(* Schneider Machine Expert - Basic project ProjectX, file version 2.7.0.0 *)
(* ProjectInformations: Name=New project *)

HARDWARE
  Cpu 0: TM221CE24U
  EthernetConfiguration: NetworkName=M221, IpAllocationMode=FixedAddress, IpAddress=0.0.0.0, SubnetMask=0.0.0.0
  SerialLineConfiguration: Baud=Baud19200, Parity=ParityEven, DataBits=DataBits8, StopBits=StopBits1, PhysicalMedium=PhysicalMediumRs485, TransmissionMode=TransmissionModeModbusRtu, SlaveId=1, Addressing=SlaveAddressing
  MastTask: UsePeriodScanMode=false, PeriodScan=100
  FastTask: Period=255
  CpuBehavior: StartingMode=StartAsPreviousState, AutoSaveRamOnEeprom=true, WatchdogPeriod=250

SYMBOLS  (address, symbol, comment, settings)
  %M240     GUI_SAFE_GUARD
  %M241     GUI_START
  %M242     GUI_ACTIVE_RESET
  %M243     GUI_SET_VALUE
  %M301     SAFE_GUARD
  %M401     INIT
  %M402     BLUE_PASS
  %M403     GREEN_PASS
  %M404     SAFETY
  %M405     INPUT
  %M406     BLUE_TANK
  %M407     EXTRA_TIME_BLUE_TANK
  %M408     GREEN_TANK
  %M409     EXTRA_TIME_GREEN_TANK
  %M410     METAL_TANK
  %M411     EXTRA_TIME_METAL_TANK
  %M412     Q_FACTOR_METAL
  %M413     Q_FACTOR_METAL_I9
  %M414     Q_FACTOR_METAL_I5
  %M415     Q_FACTOR_BLUE_I9
  %M416     Q_FACTOR_BLUE_I5
  %M417     Q_FACTOR_GREEN_I9
  %M418     Q_FACTOR_GREEN_I5
  %M421     SUS
  %M422     SUSS
  %M423     SUSSS
  %M424     SUSSSS
  %M425     SUSSSSS
  %M451     START_SYS
  %M452     STOP_SYS
  %M453     STOP_SYS_HANDLE
  %M454     STOP_SYS_HANDLE2
  %M455     CLEAR_SYS_HANDLE
  %M456     STOP_HANDLE_3
  %M457     END_SYS
  %M458     STOP_HANDLE_RESET
  %M459     HANDLE_RESET_ALL
  %M460     OVER_CONDITION
  %M461     HANDLE_CHANGE_BLUE
  %M462     HANDLE_CHANGE_BLUE2
  %M463     HANDLE_CHANGE_GREEN
  %M464     HANDLE_CHANGE_GREEN2
  %M465     HANDLE_CHANGE_METAL
  %M466     HANDLE_CHANGE_METAL2
  %M501     METAL_PART
  %M502     BLUE_LINK
  %M503     GREEN_LINK
  %M504     METAL_LINK
  %M505     SET_VALUE_LINK
  %M506     TURN_OFF_SYS
  %M507     CLEAR_SYS
  %M508     TRIGGER_TURN_OFF_SYS
  %TM0        [Preset=5, Base=OneHundredMilliSeconds]
  %TM1        [Preset=15, Base=OneHundredMilliSeconds]
  %TM2        [Preset=0, Base=OneSecond]
  %TM3        [Preset=1, Base=OneSecond]
  %TM4        [Preset=0, Base=OneSecond]
  %TM5        [Preset=1, Base=OneSecond]
  %TM6        [Preset=0, Base=OneSecond]
  %TM7        [Preset=1, Base=OneSecond]
  %TM8        [Preset=2, Base=OneSecond]
  %TM9        [Preset=2, Base=OneSecond]
  %TM10       [Preset=2, Base=OneSecond]
  %TM11       [Preset=2, Base=OneSecond]
  %TM12       [Preset=2, Base=OneSecond]
  %TM13       [Preset=2, Base=OneSecond]
  %TM14       [Preset=15, Base=OneSecond]
  %TM15       [Preset=1, Base=OneSecond]
  %TM16       [Preset=40, Base=OneSecond]
  %TM17       [Preset=3, Base=OneSecond]
  %TM18       [Preset=3, Base=OneSecond]
  %TM19       [Preset=3, Base=OneSecond]
  %TM20       [Preset=3, Base=OneSecond]
  %TM21       [Preset=3, Base=OneSecond]
  %TM22       [Preset=3, Base=OneSecond]
  %C0         "Counting"
  %C1         "Dielectric"
  %C2         "Metal"
  %C3         "Blue dielec"
  %C4         "Green dielec"
  %C5         "Blue dielec (I5)"
  %C6         "Blue dielec (I9)"
  %C7         "Green dielec (I5)"
  %C8         "Green dielec (I9)"
  %C9         "Metal (I5)"
  %C10        "Metal (I9)"
  %C11        "All time count"
  %DR0        [Bits(BitForDrum(Outputs=%M301)), StepsNumber=2]

POU New POU
  (* SectionNumber=1 *)

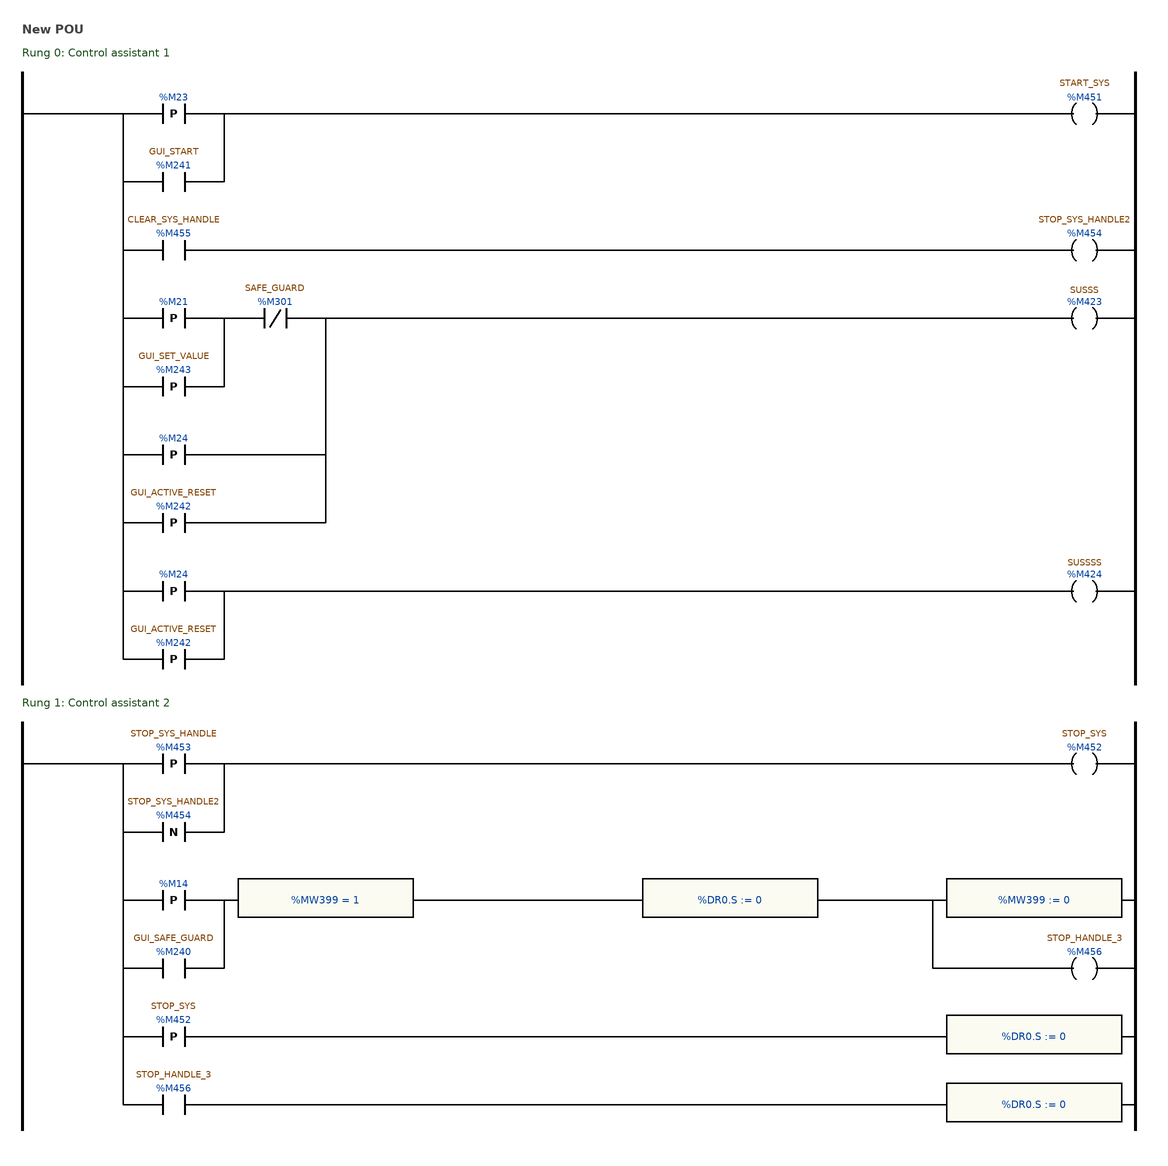

// Rung 0: Control assistant 1
  LD 1
  MPS
  AND(R %M23
  OR %M241                (* GUI_START *)
  )
  ST %M451                (* START_SYS *)
  MRD
  AND %M455               (* CLEAR_SYS_HANDLE *)
  ST %M454                (* STOP_SYS_HANDLE2 *)
  MRD
  AND(R %M21
  ORR %M243               (* GUI_SET_VALUE *)
  ANDN %M301              (* SAFE_GUARD *)
  ORR %M24
  ORR %M242               (* GUI_ACTIVE_RESET *)
  )
  ST %M423                (* SUSSS *)
  MPP
  AND(R %M24
  ORR %M242               (* GUI_ACTIVE_RESET *)
  )
  ST %M424                (* SUSSSS *)
  // as ST:
  //   START_SYS := RISING(%M23) OR GUI_START;
  //   STOP_SYS_HANDLE2 := CLEAR_SYS_HANDLE;
  //   SUSSS := (RISING(%M21) OR RISING(GUI_SET_VALUE)) AND NOT SAFE_GUARD OR RISING(%M24) OR RISING(GUI_ACTIVE_RESET);
  //   SUSSSS := RISING(%M24) OR RISING(GUI_ACTIVE_RESET);

// Rung 1: Control assistant 2
  LD 1
  MPS
  AND(R %M453             (* STOP_SYS_HANDLE *)
  ORF %M454               (* STOP_SYS_HANDLE2 *)
  )
  ST %M452                (* STOP_SYS *)
  MRD
  AND(R %M14
  OR %M240                (* GUI_SAFE_GUARD *)
  )
  AND [ %MW399 = 1 ]
  OPER [ %DR0.S := 0 ]
  [ %MW399 := 0 ]
  ST %M456                (* STOP_HANDLE_3 *)
  MRD
  ANDR %M452              (* STOP_SYS *)
  [ %DR0.S := 0 ]
  MPP
  AND %M456               (* STOP_HANDLE_3 *)
  [ %DR0.S := 0 ]
  // as ST:
  //   STOP_SYS := RISING(STOP_SYS_HANDLE) OR FALLING(STOP_SYS_HANDLE2);
  //   IF (RISING(%M14) OR GUI_SAFE_GUARD) AND %MW399 = 1 THEN %DR0.S := 0; END_IF;
  //   _t1 := (RISING(%M14) OR GUI_SAFE_GUARD) AND %MW399 = 1;
  //   IF _t1 THEN %MW399 := 0; END_IF;
  //   STOP_HANDLE_3 := _t1;
  //   IF RISING(STOP_SYS) THEN %DR0.S := 0; END_IF;
  //   IF STOP_HANDLE_3 THEN %DR0.S := 0; END_IF;

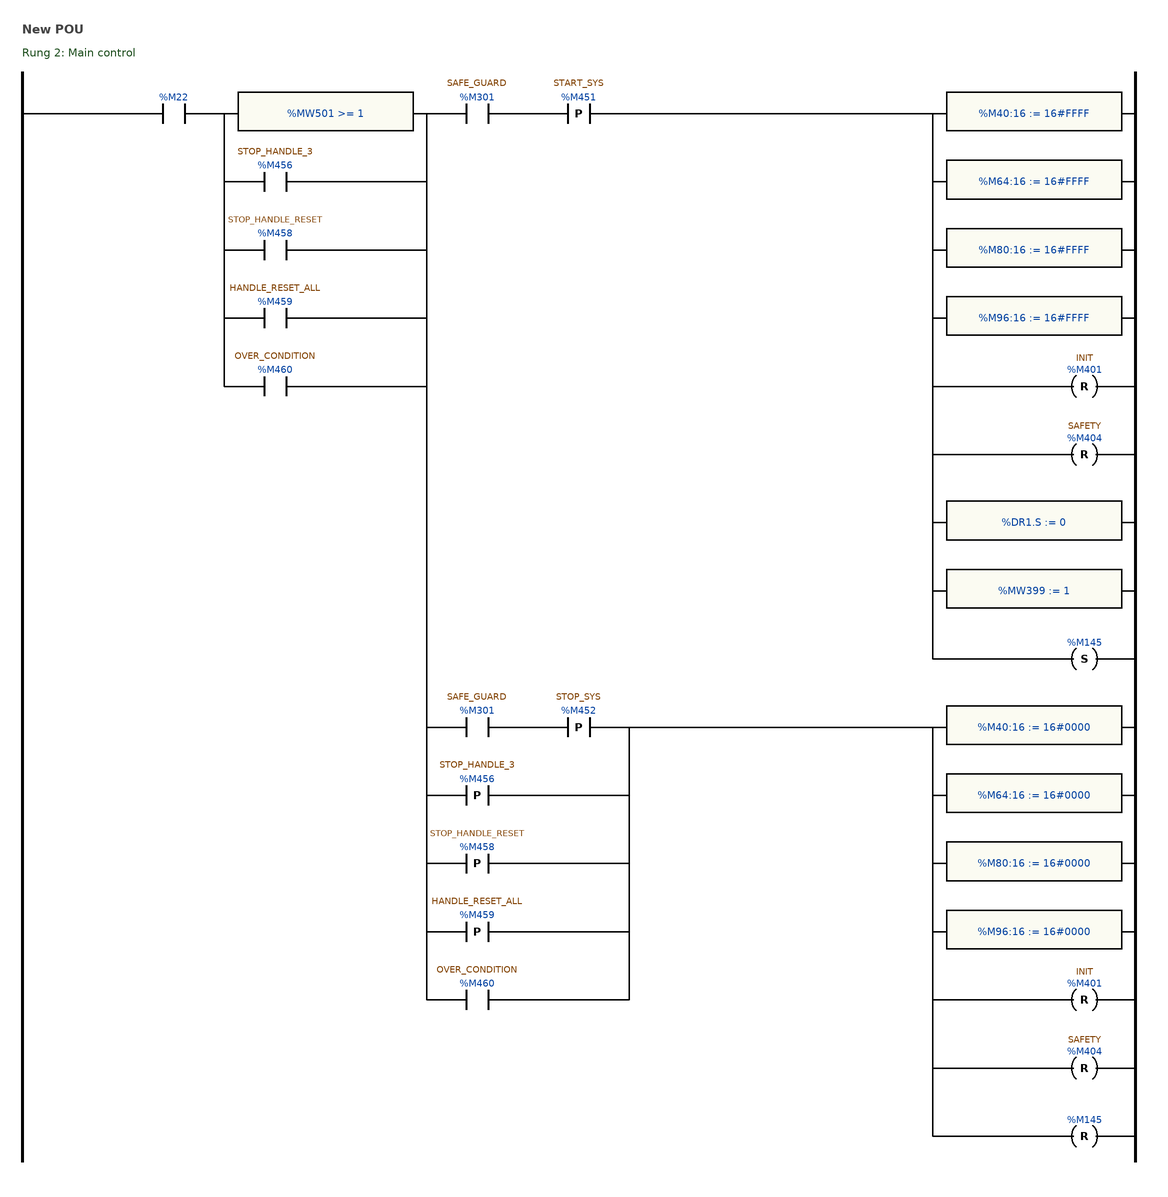

// Rung 2: Main control
  LD 1
  AND %M22
  AND( [ %MW501 >= 1 ]
  OR %M456                (* STOP_HANDLE_3 *)
  OR %M458                (* STOP_HANDLE_RESET *)
  OR %M459                (* HANDLE_RESET_ALL *)
  OR %M460                (* OVER_CONDITION *)
  )
  MPS
  AND %M301               (* SAFE_GUARD *)
  ANDR %M451              (* START_SYS *)
  [ %M40:16 := 16#FFFF ]
  [ %M64:16 := 16#FFFF ]
  [ %M80:16 := 16#FFFF ]
  [ %M96:16 := 16#FFFF ]
  R %M401                 (* INIT *)
  R %M404                 (* SAFETY *)
  [ %DR1.S := 0 ]
  [ %MW399 := 1 ]
  S %M145
  MPP
  AND( %M301              (* SAFE_GUARD *)
  ANDR %M452              (* STOP_SYS *)
  ORR %M456               (* STOP_HANDLE_3 *)
  ORR %M458               (* STOP_HANDLE_RESET *)
  ORR %M459               (* HANDLE_RESET_ALL *)
  OR %M460                (* OVER_CONDITION *)
  )
  [ %M40:16 := 16#0000 ]
  [ %M64:16 := 16#0000 ]
  [ %M80:16 := 16#0000 ]
  [ %M96:16 := 16#0000 ]
  R %M401                 (* INIT *)
  R %M404                 (* SAFETY *)
  R %M145
  // as ST:
  //   IF %M22 AND (%MW501 >= 1 OR STOP_HANDLE_3 OR STOP_HANDLE_RESET OR HANDLE_RESET_ALL OR OVER_CONDITION) AND SAFE_GUARD AND RISING(START_SYS) THEN %M40:16 := 16#FFFF; END_IF;
  //   IF %M22 AND (%MW501 >= 1 OR STOP_HANDLE_3 OR STOP_HANDLE_RESET OR HANDLE_RESET_ALL OR OVER_CONDITION) AND SAFE_GUARD AND RISING(START_SYS) THEN %M64:16 := 16#FFFF; END_IF;
  //   IF %M22 AND (%MW501 >= 1 OR STOP_HANDLE_3 OR STOP_HANDLE_RESET OR HANDLE_RESET_ALL OR OVER_CONDITION) AND SAFE_GUARD AND RISING(START_SYS) THEN %M80:16 := 16#FFFF; END_IF;
  //   IF %M22 AND (%MW501 >= 1 OR STOP_HANDLE_3 OR STOP_HANDLE_RESET OR HANDLE_RESET_ALL OR OVER_CONDITION) AND SAFE_GUARD AND RISING(START_SYS) THEN %M96:16 := 16#FFFF; END_IF;
  //   IF %M22 AND (%MW501 >= 1 OR STOP_HANDLE_3 OR STOP_HANDLE_RESET OR HANDLE_RESET_ALL OR OVER_CONDITION) AND SAFE_GUARD AND RISING(START_SYS) THEN INIT := FALSE; END_IF;
  //   IF %M22 AND (%MW501 >= 1 OR STOP_HANDLE_3 OR STOP_HANDLE_RESET OR HANDLE_RESET_ALL OR OVER_CONDITION) AND SAFE_GUARD AND RISING(START_SYS) THEN SAFETY := FALSE; END_IF;
  //   IF %M22 AND (%MW501 >= 1 OR STOP_HANDLE_3 OR STOP_HANDLE_RESET OR HANDLE_RESET_ALL OR OVER_CONDITION) AND SAFE_GUARD AND RISING(START_SYS) THEN %DR1.S := 0; END_IF;
  //   IF %M22 AND (%MW501 >= 1 OR STOP_HANDLE_3 OR STOP_HANDLE_RESET OR HANDLE_RESET_ALL OR OVER_CONDITION) AND SAFE_GUARD AND RISING(START_SYS) THEN %MW399 := 1; END_IF;
  //   IF %M22 AND (%MW501 >= 1 OR STOP_HANDLE_3 OR STOP_HANDLE_RESET OR HANDLE_RESET_ALL OR OVER_CONDITION) AND SAFE_GUARD AND RISING(START_SYS) THEN %M145 := TRUE; END_IF;
  //   IF %M22 AND (%MW501 >= 1 OR STOP_HANDLE_3 OR STOP_HANDLE_RESET OR HANDLE_RESET_ALL OR OVER_CONDITION) AND (SAFE_GUARD AND RISING(STOP_SYS) OR RISING(STOP_HANDLE_3) OR RISING(STOP_HANDLE_RESET) OR RISING(HANDLE_RESET_ALL) OR OVER_CONDITION) THEN %M40:16 := 16#0000; END_IF;
  //   IF %M22 AND (%MW501 >= 1 OR STOP_HANDLE_3 OR STOP_HANDLE_RESET OR HANDLE_RESET_ALL OR OVER_CONDITION) AND (SAFE_GUARD AND RISING(STOP_SYS) OR RISING(STOP_HANDLE_3) OR RISING(STOP_HANDLE_RESET) OR RISING(HANDLE_RESET_ALL) OR OVER_CONDITION) THEN %M64:16 := 16#0000; END_IF;
  //   IF %M22 AND (%MW501 >= 1 OR STOP_HANDLE_3 OR STOP_HANDLE_RESET OR HANDLE_RESET_ALL OR OVER_CONDITION) AND (SAFE_GUARD AND RISING(STOP_SYS) OR RISING(STOP_HANDLE_3) OR RISING(STOP_HANDLE_RESET) OR RISING(HANDLE_RESET_ALL) OR OVER_CONDITION) THEN %M80:16 := 16#0000; END_IF;
  //   IF %M22 AND (%MW501 >= 1 OR STOP_HANDLE_3 OR STOP_HANDLE_RESET OR HANDLE_RESET_ALL OR OVER_CONDITION) AND (SAFE_GUARD AND RISING(STOP_SYS) OR RISING(STOP_HANDLE_3) OR RISING(STOP_HANDLE_RESET) OR RISING(HANDLE_RESET_ALL) OR OVER_CONDITION) THEN %M96:16 := 16#0000; END_IF;
  //   IF %M22 AND (%MW501 >= 1 OR STOP_HANDLE_3 OR STOP_HANDLE_RESET OR HANDLE_RESET_ALL OR OVER_CONDITION) AND (SAFE_GUARD AND RISING(STOP_SYS) OR RISING(STOP_HANDLE_3) OR RISING(STOP_HANDLE_RESET) OR RISING(HANDLE_RESET_ALL) OR OVER_CONDITION) THEN INIT := FALSE; END_IF;
  //   IF %M22 AND (%MW501 >= 1 OR STOP_HANDLE_3 OR STOP_HANDLE_RESET OR HANDLE_RESET_ALL OR OVER_CONDITION) AND (SAFE_GUARD AND RISING(STOP_SYS) OR RISING(STOP_HANDLE_3) OR RISING(STOP_HANDLE_RESET) OR RISING(HANDLE_RESET_ALL) OR OVER_CONDITION) THEN SAFETY := FALSE; END_IF;
  //   IF %M22 AND (%MW501 >= 1 OR STOP_HANDLE_3 OR STOP_HANDLE_RESET OR HANDLE_RESET_ALL OR OVER_CONDITION) AND (SAFE_GUARD AND RISING(STOP_SYS) OR RISING(STOP_HANDLE_3) OR RISING(STOP_HANDLE_RESET) OR RISING(HANDLE_RESET_ALL) OR OVER_CONDITION) THEN %M145 := FALSE; END_IF;

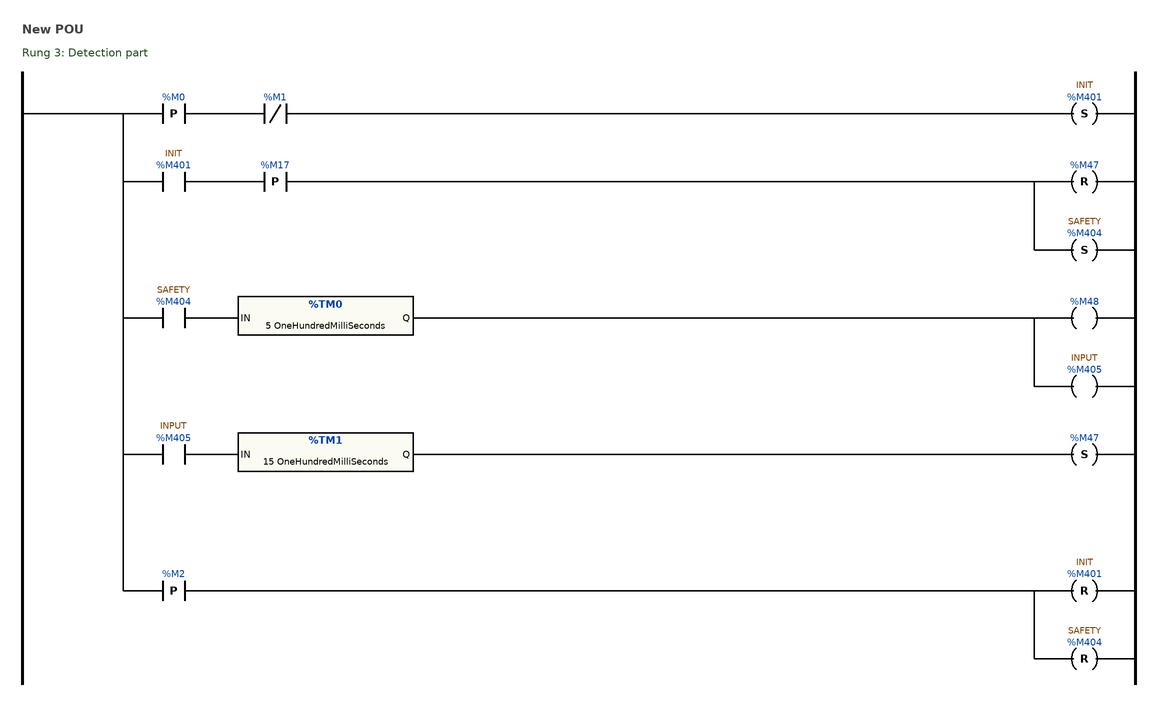

// Rung 3: Detection part
  LD 1
  MULTIFB
  LD 1
  ST %MW2009:X0
  LD %MW2009:X0
  MPS
  ANDR %M0
  ANDN %M1
  S %M401                 (* INIT *)
  MPP
  AND %M401               (* INIT *)
  ANDR %M17
  R %M47
  S %M404                 (* SAFETY *)
  BLK %TM0
  LD %MW2009:X0
  AND %M404               (* SAFETY *)
  IN
  OUT_BLK
  LD Q
  ST %M48
  ST %M405                (* INPUT *)
  END_BLK
  BLK %TM1
  LD %MW2009:X0
  AND %M405               (* INPUT *)
  IN
  OUT_BLK
  LD Q
  S %M47
  END_BLK
  LD %MW2009:X0
  ANDR %M2
  R %M401                 (* INIT *)
  R %M404                 (* SAFETY *)
  MULTIFB
  // as ST:
  //   IF RISING(%M0) AND NOT %M1 THEN INIT := TRUE; END_IF;
  //   IF INIT AND RISING(%M17) THEN %M47 := FALSE; END_IF;
  //   IF INIT AND RISING(%M17) THEN SAFETY := TRUE; END_IF;
  //   %TM0(IN := SAFETY);
  //   %M48 := %TM0.Q;
  //   INPUT := %TM0.Q;
  //   %TM1(IN := INPUT);
  //   IF %TM1.Q THEN %M47 := TRUE; END_IF;
  //   IF RISING(%M2) THEN INIT := FALSE; END_IF;
  //   IF RISING(%M2) THEN SAFETY := FALSE; END_IF;

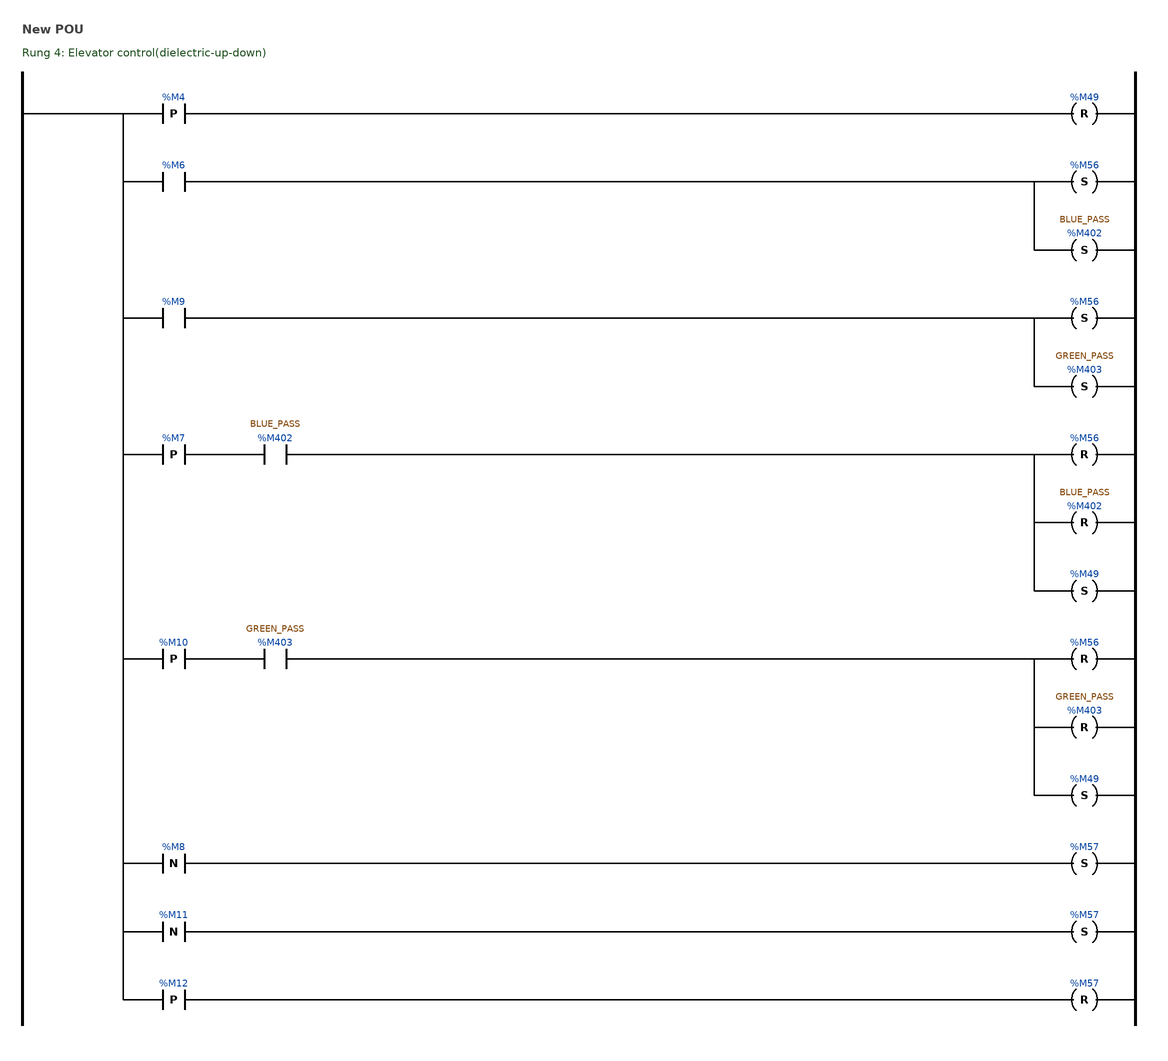

// Rung 4: Elevator control(dielectric-up-down)
  LD 1
  MPS
  ANDR %M4
  R %M49
  MRD
  AND %M6
  S %M56
  S %M402                 (* BLUE_PASS *)
  MRD
  AND %M9
  S %M56
  S %M403                 (* GREEN_PASS *)
  MRD
  ANDR %M7
  AND %M402               (* BLUE_PASS *)
  R %M56
  R %M402                 (* BLUE_PASS *)
  S %M49
  MRD
  ANDR %M10
  AND %M403               (* GREEN_PASS *)
  R %M56
  R %M403                 (* GREEN_PASS *)
  S %M49
  MRD
  ANDF %M8
  S %M57
  MRD
  ANDF %M11
  S %M57
  MPP
  ANDR %M12
  R %M57
  // as ST:
  //   IF RISING(%M4) THEN %M49 := FALSE; END_IF;
  //   IF %M6 THEN %M56 := TRUE; END_IF;
  //   IF %M6 THEN BLUE_PASS := TRUE; END_IF;
  //   IF %M9 THEN %M56 := TRUE; END_IF;
  //   IF %M9 THEN GREEN_PASS := TRUE; END_IF;
  //   IF RISING(%M7) AND BLUE_PASS THEN %M56 := FALSE; END_IF;
  //   _t1 := RISING(%M7) AND BLUE_PASS;
  //   IF _t1 THEN BLUE_PASS := FALSE; END_IF;
  //   IF _t1 THEN %M49 := TRUE; END_IF;
  //   IF RISING(%M10) AND GREEN_PASS THEN %M56 := FALSE; END_IF;
  //   _t2 := RISING(%M10) AND GREEN_PASS;
  //   IF _t2 THEN GREEN_PASS := FALSE; END_IF;
  //   IF _t2 THEN %M49 := TRUE; END_IF;
  //   IF FALLING(%M8) THEN %M57 := TRUE; END_IF;
  //   IF FALLING(%M11) THEN %M57 := TRUE; END_IF;
  //   IF RISING(%M12) THEN %M57 := FALSE; END_IF;

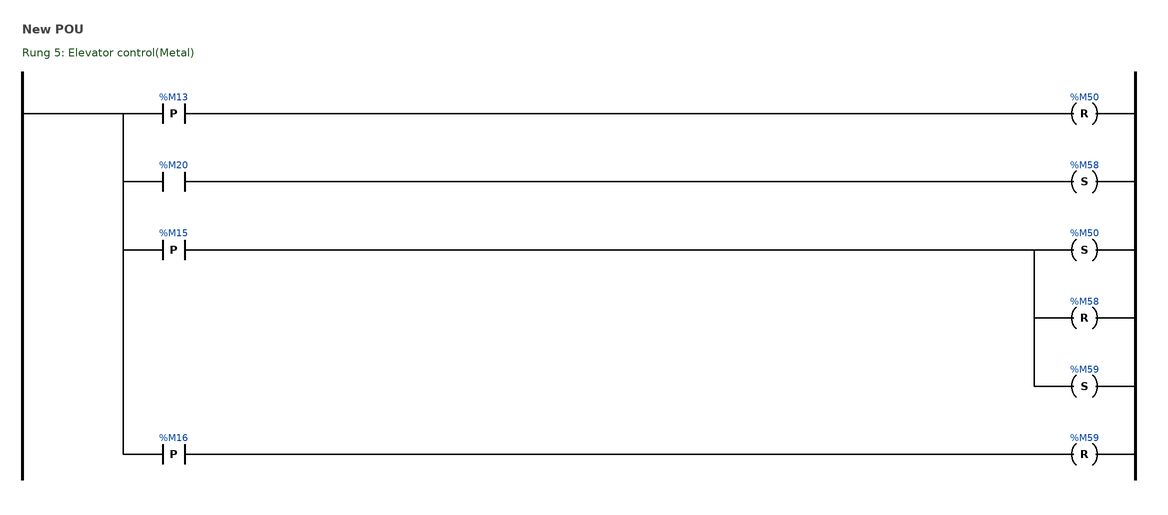

// Rung 5: Elevator control(Metal)
  LD 1
  MPS
  ANDR %M13
  R %M50
  MRD
  AND %M20
  S %M58
  MRD
  ANDR %M15
  S %M50
  R %M58
  S %M59
  MPP
  ANDR %M16
  R %M59
  // as ST:
  //   IF RISING(%M13) THEN %M50 := FALSE; END_IF;
  //   IF %M20 THEN %M58 := TRUE; END_IF;
  //   IF RISING(%M15) THEN %M50 := TRUE; END_IF;
  //   IF RISING(%M15) THEN %M58 := FALSE; END_IF;
  //   IF RISING(%M15) THEN %M59 := TRUE; END_IF;
  //   IF RISING(%M16) THEN %M59 := FALSE; END_IF;

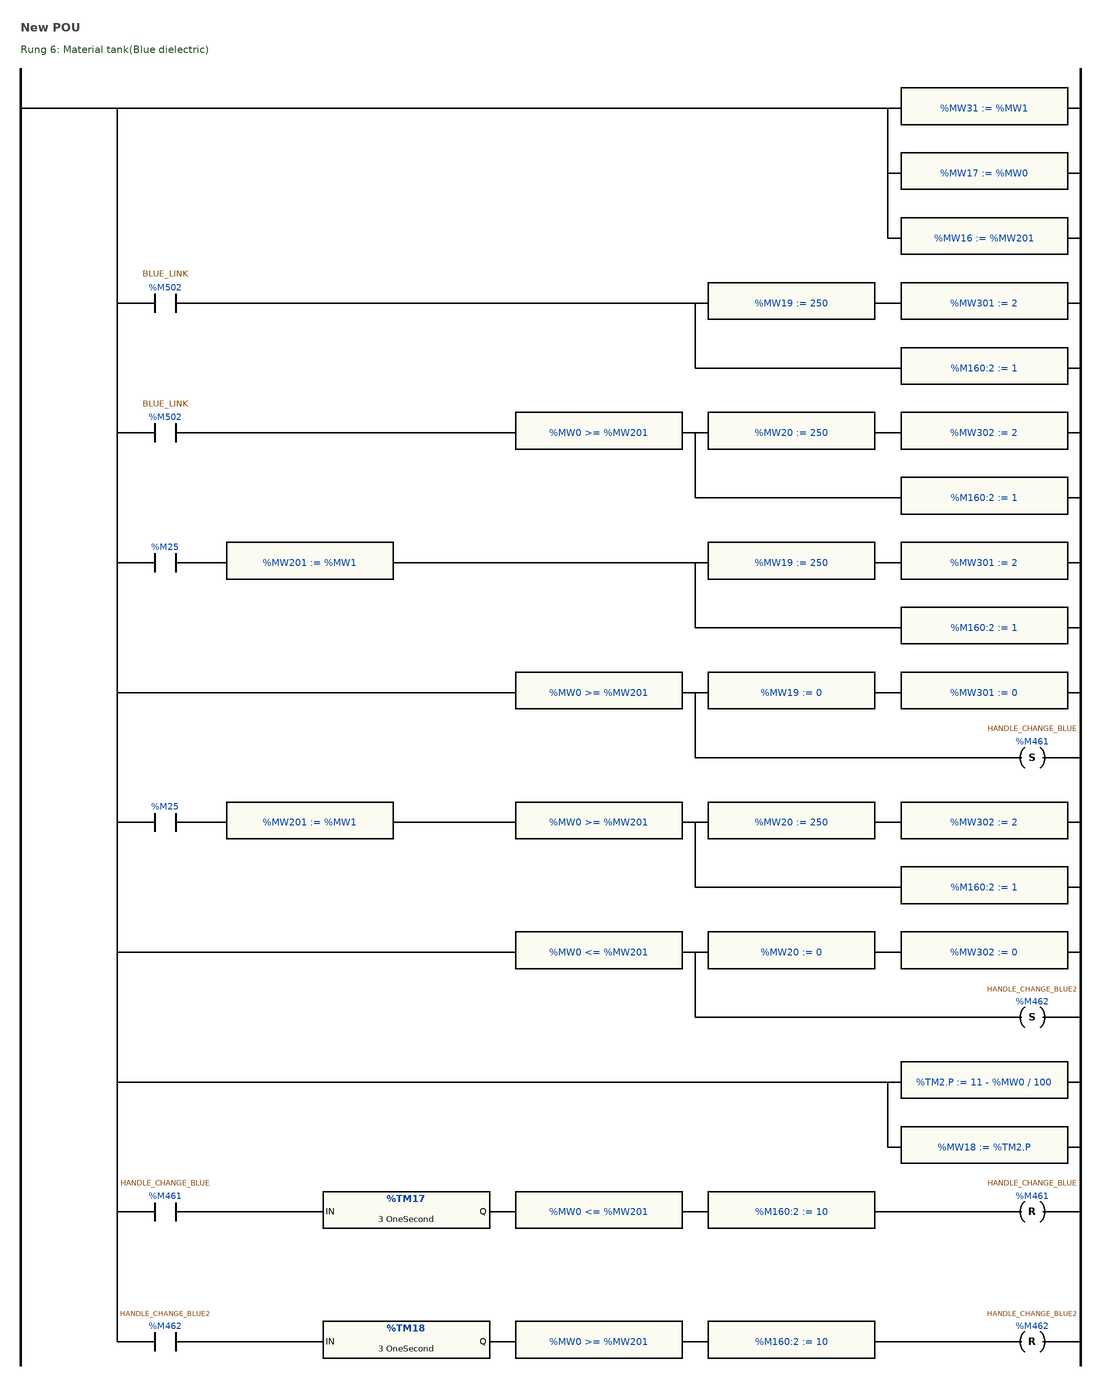

// Rung 6: Material tank(Blue dielectric)
  LD 1
  MULTIFB
  LD 1
  ST %MW2009:X0
  LD %MW2009:X0
  MPS
  [ %MW31 := %MW1 ]
  [ %MW17 := %MW0 ]
  [ %MW16 := %MW201 ]
  MRD
  AND %M502               (* BLUE_LINK *)
  MPS
  OPER [ %MW19 := 250 ]
  [ %MW301 := 2 ]
  MPP
  [ %M160:2 := 1 ]
  MRD
  AND %M502               (* BLUE_LINK *)
  AND [ %MW0 >= %MW201 ]
  MPS
  OPER [ %MW20 := 250 ]
  [ %MW302 := 2 ]
  MPP
  [ %M160:2 := 1 ]
  MRD
  AND %M25
  OPER [ %MW201 := %MW1 ]
  MPS
  OPER [ %MW19 := 250 ]
  [ %MW301 := 2 ]
  MPP
  [ %M160:2 := 1 ]
  MRD
  AND [ %MW0 >= %MW201 ]
  MPS
  OPER [ %MW19 := 0 ]
  [ %MW301 := 0 ]
  MPP
  S %M461                 (* HANDLE_CHANGE_BLUE *)
  MRD
  AND %M25
  OPER [ %MW201 := %MW1 ]
  AND [ %MW0 >= %MW201 ]
  MPS
  OPER [ %MW20 := 250 ]
  [ %MW302 := 2 ]
  MPP
  [ %M160:2 := 1 ]
  MRD
  AND [ %MW0 <= %MW201 ]
  MPS
  OPER [ %MW20 := 0 ]
  [ %MW302 := 0 ]
  MPP
  S %M462                 (* HANDLE_CHANGE_BLUE2 *)
  MPP
  [ %TM2.P := 11 - %MW0 / 100 ]
  [ %MW18 := %TM2.P ]
  BLK %TM17
  LD %MW2009:X0
  AND %M461               (* HANDLE_CHANGE_BLUE *)
  IN
  OUT_BLK
  LD Q
  AND [ %MW0 <= %MW201 ]
  OPER [ %M160:2 := 10 ]
  R %M461                 (* HANDLE_CHANGE_BLUE *)
  END_BLK
  BLK %TM18
  LD %MW2009:X0
  AND %M462               (* HANDLE_CHANGE_BLUE2 *)
  IN
  OUT_BLK
  LD Q
  AND [ %MW0 >= %MW201 ]
  OPER [ %M160:2 := 10 ]
  R %M462                 (* HANDLE_CHANGE_BLUE2 *)
  END_BLK
  MULTIFB
  // as ST:
  //   %MW31 := %MW1;
  //   %MW17 := %MW0;
  //   %MW16 := %MW201;
  //   IF BLUE_LINK THEN %MW19 := 250; END_IF;
  //   IF BLUE_LINK THEN %MW301 := 2; END_IF;
  //   IF BLUE_LINK THEN %M160:2 := 1; END_IF;
  //   IF BLUE_LINK AND %MW0 >= %MW201 THEN %MW20 := 250; END_IF;
  //   IF BLUE_LINK AND %MW0 >= %MW201 THEN %MW302 := 2; END_IF;
  //   IF BLUE_LINK AND %MW0 >= %MW201 THEN %M160:2 := 1; END_IF;
  //   IF %M25 THEN %MW201 := %MW1; END_IF;
  //   IF %M25 THEN %MW19 := 250; END_IF;
  //   IF %M25 THEN %MW301 := 2; END_IF;
  //   IF %M25 THEN %M160:2 := 1; END_IF;
  //   IF %MW0 >= %MW201 THEN %MW19 := 0; END_IF;
  //   IF %MW0 >= %MW201 THEN %MW301 := 0; END_IF;
  //   IF %MW0 >= %MW201 THEN HANDLE_CHANGE_BLUE := TRUE; END_IF;
  //   IF %M25 THEN %MW201 := %MW1; END_IF;
  //   IF %M25 AND %MW0 >= %MW201 THEN %MW20 := 250; END_IF;
  //   IF %M25 AND %MW0 >= %MW201 THEN %MW302 := 2; END_IF;
  //   IF %M25 AND %MW0 >= %MW201 THEN %M160:2 := 1; END_IF;
  //   IF %MW0 <= %MW201 THEN %MW20 := 0; END_IF;
  //   IF %MW0 <= %MW201 THEN %MW302 := 0; END_IF;
  //   IF %MW0 <= %MW201 THEN HANDLE_CHANGE_BLUE2 := TRUE; END_IF;
  //   %TM2.P := 11 - %MW0 / 100;
  //   %MW18 := %TM2.P;
  //   %TM17(IN := HANDLE_CHANGE_BLUE);
  //   IF %TM17.Q AND %MW0 <= %MW201 THEN %M160:2 := 10; END_IF;
  //   IF %TM17.Q AND %MW0 <= %MW201 THEN HANDLE_CHANGE_BLUE := FALSE; END_IF;
  //   %TM18(IN := HANDLE_CHANGE_BLUE2);
  //   IF %TM18.Q AND %MW0 >= %MW201 THEN %M160:2 := 10; END_IF;
  //   IF %TM18.Q AND %MW0 >= %MW201 THEN HANDLE_CHANGE_BLUE2 := FALSE; END_IF;

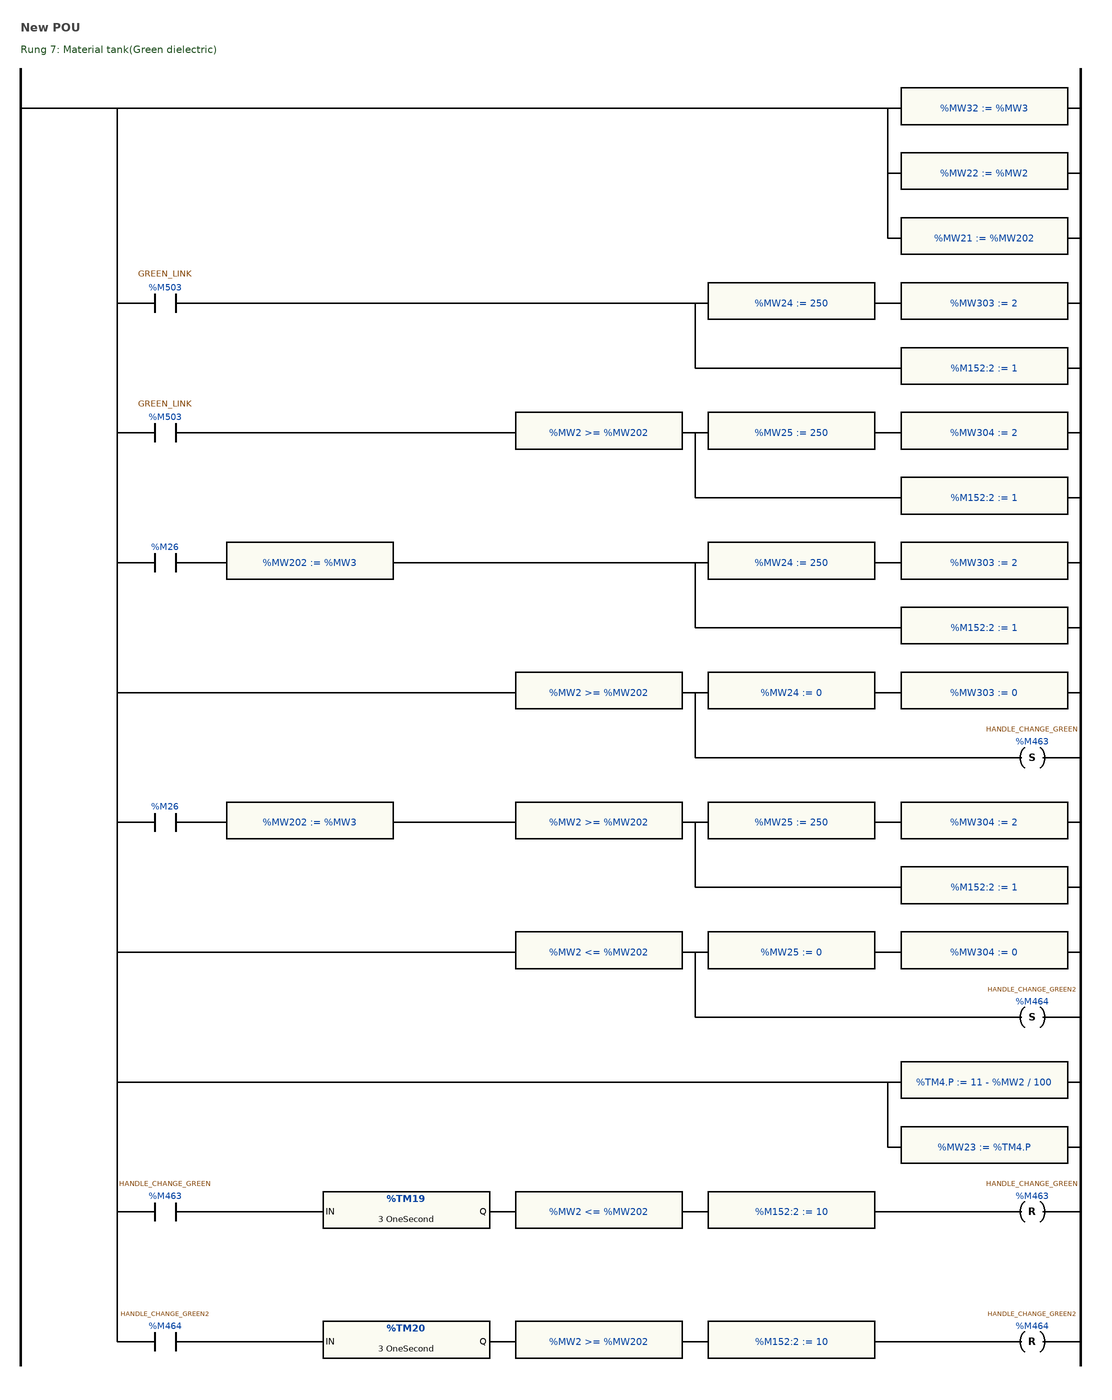

// Rung 7: Material tank(Green dielectric)
  LD 1
  MULTIFB
  LD 1
  ST %MW2009:X0
  LD %MW2009:X0
  MPS
  [ %MW32 := %MW3 ]
  [ %MW22 := %MW2 ]
  [ %MW21 := %MW202 ]
  MRD
  AND %M503               (* GREEN_LINK *)
  MPS
  OPER [ %MW24 := 250 ]
  [ %MW303 := 2 ]
  MPP
  [ %M152:2 := 1 ]
  MRD
  AND %M503               (* GREEN_LINK *)
  AND [ %MW2 >= %MW202 ]
  MPS
  OPER [ %MW25 := 250 ]
  [ %MW304 := 2 ]
  MPP
  [ %M152:2 := 1 ]
  MRD
  AND %M26
  OPER [ %MW202 := %MW3 ]
  MPS
  OPER [ %MW24 := 250 ]
  [ %MW303 := 2 ]
  MPP
  [ %M152:2 := 1 ]
  MRD
  AND [ %MW2 >= %MW202 ]
  MPS
  OPER [ %MW24 := 0 ]
  [ %MW303 := 0 ]
  MPP
  S %M463                 (* HANDLE_CHANGE_GREEN *)
  MRD
  AND %M26
  OPER [ %MW202 := %MW3 ]
  AND [ %MW2 >= %MW202 ]
  MPS
  OPER [ %MW25 := 250 ]
  [ %MW304 := 2 ]
  MPP
  [ %M152:2 := 1 ]
  MRD
  AND [ %MW2 <= %MW202 ]
  MPS
  OPER [ %MW25 := 0 ]
  [ %MW304 := 0 ]
  MPP
  S %M464                 (* HANDLE_CHANGE_GREEN2 *)
  MPP
  [ %TM4.P := 11 - %MW2 / 100 ]
  [ %MW23 := %TM4.P ]
  BLK %TM19
  LD %MW2009:X0
  AND %M463               (* HANDLE_CHANGE_GREEN *)
  IN
  OUT_BLK
  LD Q
  AND [ %MW2 <= %MW202 ]
  OPER [ %M152:2 := 10 ]
  R %M463                 (* HANDLE_CHANGE_GREEN *)
  END_BLK
  BLK %TM20
  LD %MW2009:X0
  AND %M464               (* HANDLE_CHANGE_GREEN2 *)
  IN
  OUT_BLK
  LD Q
  AND [ %MW2 >= %MW202 ]
  OPER [ %M152:2 := 10 ]
  R %M464                 (* HANDLE_CHANGE_GREEN2 *)
  END_BLK
  MULTIFB
  // as ST:
  //   %MW32 := %MW3;
  //   %MW22 := %MW2;
  //   %MW21 := %MW202;
  //   IF GREEN_LINK THEN %MW24 := 250; END_IF;
  //   IF GREEN_LINK THEN %MW303 := 2; END_IF;
  //   IF GREEN_LINK THEN %M152:2 := 1; END_IF;
  //   IF GREEN_LINK AND %MW2 >= %MW202 THEN %MW25 := 250; END_IF;
  //   IF GREEN_LINK AND %MW2 >= %MW202 THEN %MW304 := 2; END_IF;
  //   IF GREEN_LINK AND %MW2 >= %MW202 THEN %M152:2 := 1; END_IF;
  //   IF %M26 THEN %MW202 := %MW3; END_IF;
  //   IF %M26 THEN %MW24 := 250; END_IF;
  //   IF %M26 THEN %MW303 := 2; END_IF;
  //   IF %M26 THEN %M152:2 := 1; END_IF;
  //   IF %MW2 >= %MW202 THEN %MW24 := 0; END_IF;
  //   IF %MW2 >= %MW202 THEN %MW303 := 0; END_IF;
  //   IF %MW2 >= %MW202 THEN HANDLE_CHANGE_GREEN := TRUE; END_IF;
  //   IF %M26 THEN %MW202 := %MW3; END_IF;
  //   IF %M26 AND %MW2 >= %MW202 THEN %MW25 := 250; END_IF;
  //   IF %M26 AND %MW2 >= %MW202 THEN %MW304 := 2; END_IF;
  //   IF %M26 AND %MW2 >= %MW202 THEN %M152:2 := 1; END_IF;
  //   IF %MW2 <= %MW202 THEN %MW25 := 0; END_IF;
  //   IF %MW2 <= %MW202 THEN %MW304 := 0; END_IF;
  //   IF %MW2 <= %MW202 THEN HANDLE_CHANGE_GREEN2 := TRUE; END_IF;
  //   %TM4.P := 11 - %MW2 / 100;
  //   %MW23 := %TM4.P;
  //   %TM19(IN := HANDLE_CHANGE_GREEN);
  //   IF %TM19.Q AND %MW2 <= %MW202 THEN %M152:2 := 10; END_IF;
  //   IF %TM19.Q AND %MW2 <= %MW202 THEN HANDLE_CHANGE_GREEN := FALSE; END_IF;
  //   %TM20(IN := HANDLE_CHANGE_GREEN2);
  //   IF %TM20.Q AND %MW2 >= %MW202 THEN %M152:2 := 10; END_IF;
  //   IF %TM20.Q AND %MW2 >= %MW202 THEN HANDLE_CHANGE_GREEN2 := FALSE; END_IF;

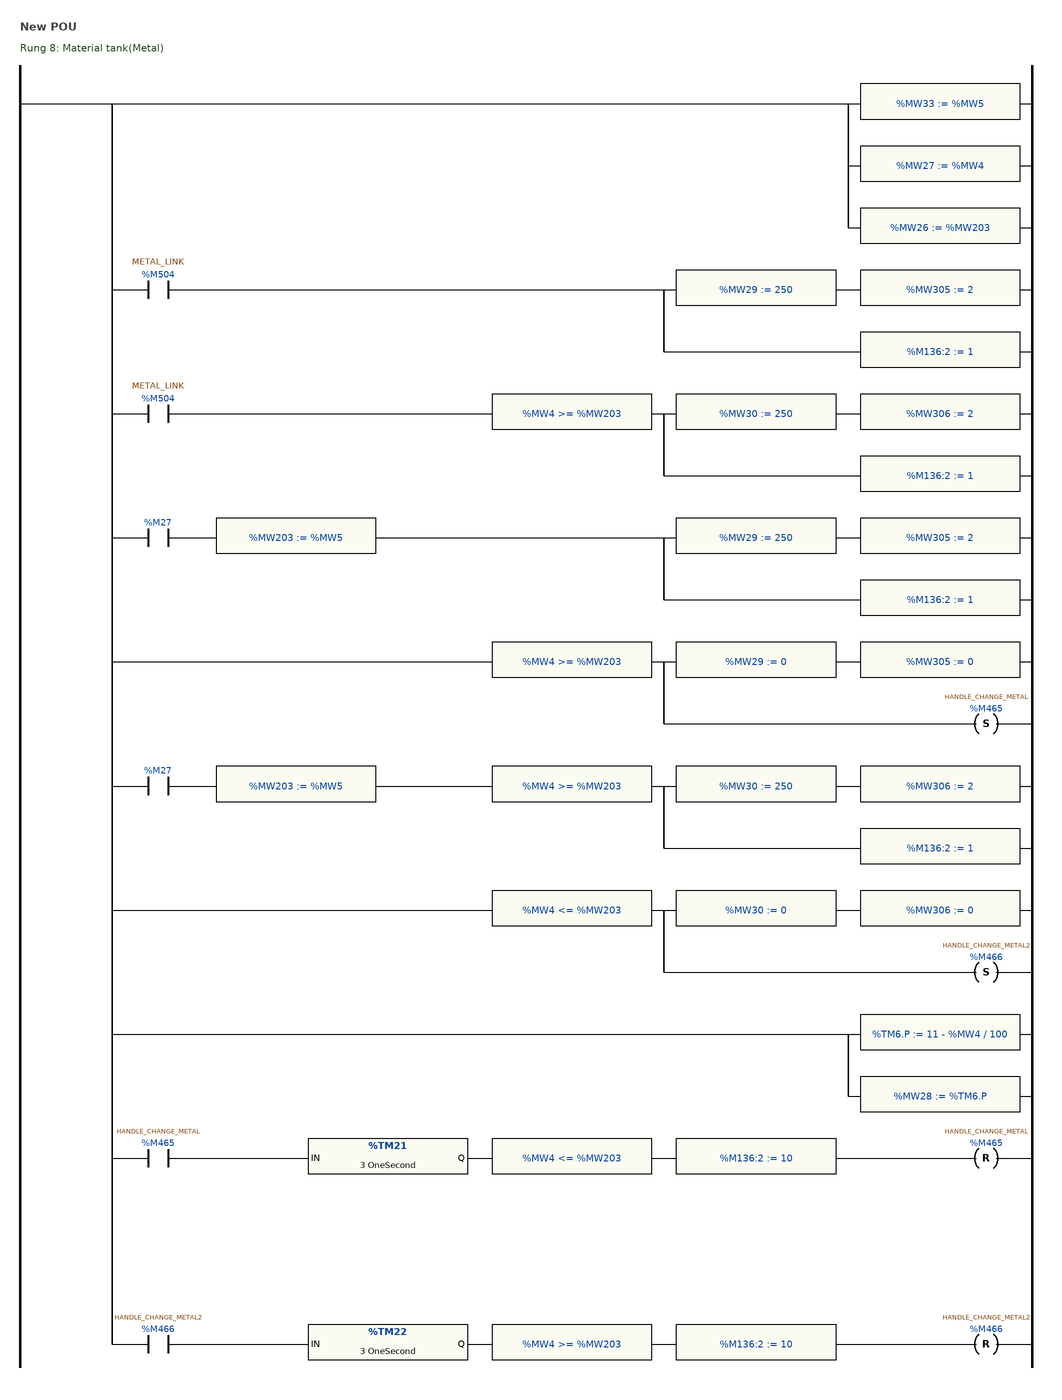

// Rung 8: Material tank(Metal)
  LD 1
  MULTIFB
  LD 1
  ST %MW2009:X0
  LD %MW2009:X0
  MPS
  [ %MW33 := %MW5 ]
  [ %MW27 := %MW4 ]
  [ %MW26 := %MW203 ]
  MRD
  AND %M504               (* METAL_LINK *)
  MPS
  OPER [ %MW29 := 250 ]
  [ %MW305 := 2 ]
  MPP
  [ %M136:2 := 1 ]
  MRD
  AND %M504               (* METAL_LINK *)
  AND [ %MW4 >= %MW203 ]
  MPS
  OPER [ %MW30 := 250 ]
  [ %MW306 := 2 ]
  MPP
  [ %M136:2 := 1 ]
  MRD
  AND %M27
  OPER [ %MW203 := %MW5 ]
  MPS
  OPER [ %MW29 := 250 ]
  [ %MW305 := 2 ]
  MPP
  [ %M136:2 := 1 ]
  MRD
  AND [ %MW4 >= %MW203 ]
  MPS
  OPER [ %MW29 := 0 ]
  [ %MW305 := 0 ]
  MPP
  S %M465                 (* HANDLE_CHANGE_METAL *)
  MRD
  AND %M27
  OPER [ %MW203 := %MW5 ]
  AND [ %MW4 >= %MW203 ]
  MPS
  OPER [ %MW30 := 250 ]
  [ %MW306 := 2 ]
  MPP
  [ %M136:2 := 1 ]
  MRD
  AND [ %MW4 <= %MW203 ]
  MPS
  OPER [ %MW30 := 0 ]
  [ %MW306 := 0 ]
  MPP
  S %M466                 (* HANDLE_CHANGE_METAL2 *)
  MPP
  [ %TM6.P := 11 - %MW4 / 100 ]
  [ %MW28 := %TM6.P ]
  BLK %TM21
  LD %MW2009:X0
  AND %M465               (* HANDLE_CHANGE_METAL *)
  IN
  OUT_BLK
  LD Q
  AND [ %MW4 <= %MW203 ]
  OPER [ %M136:2 := 10 ]
  R %M465                 (* HANDLE_CHANGE_METAL *)
  END_BLK
  BLK %TM22
  LD %MW2009:X0
  AND %M466               (* HANDLE_CHANGE_METAL2 *)
  IN
  OUT_BLK
  LD Q
  AND [ %MW4 >= %MW203 ]
  OPER [ %M136:2 := 10 ]
  R %M466                 (* HANDLE_CHANGE_METAL2 *)
  END_BLK
  MULTIFB
  // as ST:
  //   %MW33 := %MW5;
  //   %MW27 := %MW4;
  //   %MW26 := %MW203;
  //   IF METAL_LINK THEN %MW29 := 250; END_IF;
  //   IF METAL_LINK THEN %MW305 := 2; END_IF;
  //   IF METAL_LINK THEN %M136:2 := 1; END_IF;
  //   IF METAL_LINK AND %MW4 >= %MW203 THEN %MW30 := 250; END_IF;
  //   IF METAL_LINK AND %MW4 >= %MW203 THEN %MW306 := 2; END_IF;
  //   IF METAL_LINK AND %MW4 >= %MW203 THEN %M136:2 := 1; END_IF;
  //   IF %M27 THEN %MW203 := %MW5; END_IF;
  //   IF %M27 THEN %MW29 := 250; END_IF;
  //   IF %M27 THEN %MW305 := 2; END_IF;
  //   IF %M27 THEN %M136:2 := 1; END_IF;
  //   IF %MW4 >= %MW203 THEN %MW29 := 0; END_IF;
  //   IF %MW4 >= %MW203 THEN %MW305 := 0; END_IF;
  //   IF %MW4 >= %MW203 THEN HANDLE_CHANGE_METAL := TRUE; END_IF;
  //   IF %M27 THEN %MW203 := %MW5; END_IF;
  //   IF %M27 AND %MW4 >= %MW203 THEN %MW30 := 250; END_IF;
  //   IF %M27 AND %MW4 >= %MW203 THEN %MW306 := 2; END_IF;
  //   IF %M27 AND %MW4 >= %MW203 THEN %M136:2 := 1; END_IF;
  //   IF %MW4 <= %MW203 THEN %MW30 := 0; END_IF;
  //   IF %MW4 <= %MW203 THEN %MW306 := 0; END_IF;
  //   IF %MW4 <= %MW203 THEN HANDLE_CHANGE_METAL2 := TRUE; END_IF;
  //   %TM6.P := 11 - %MW4 / 100;
  //   %MW28 := %TM6.P;
  //   %TM21(IN := HANDLE_CHANGE_METAL);
  //   IF %TM21.Q AND %MW4 <= %MW203 THEN %M136:2 := 10; END_IF;
  //   IF %TM21.Q AND %MW4 <= %MW203 THEN HANDLE_CHANGE_METAL := FALSE; END_IF;
  //   %TM22(IN := HANDLE_CHANGE_METAL2);
  //   IF %TM22.Q AND %MW4 >= %MW203 THEN %M136:2 := 10; END_IF;
  //   IF %TM22.Q AND %MW4 >= %MW203 THEN HANDLE_CHANGE_METAL2 := FALSE; END_IF;

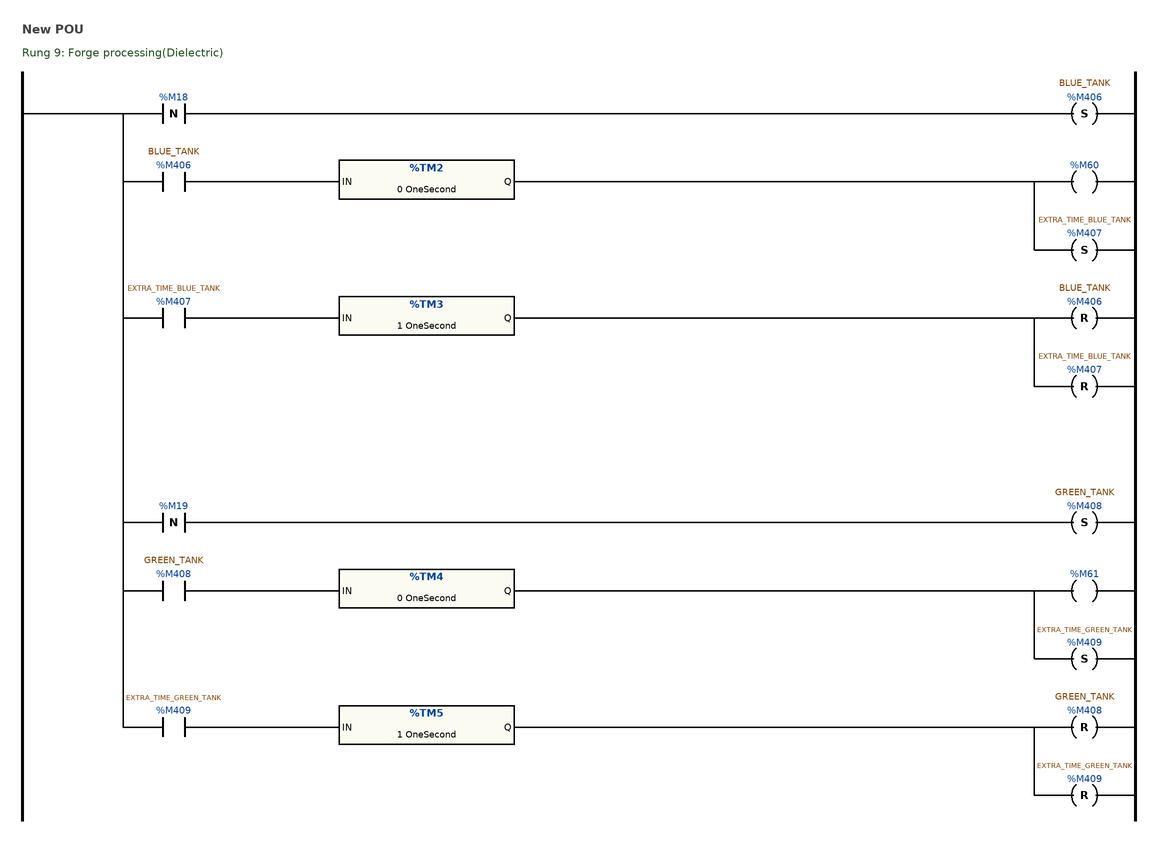

// Rung 9: Forge processing(Dielectric)
  LD 1
  MULTIFB
  LD 1
  ST %MW2009:X0
  LD %MW2009:X0
  ANDF %M18
  S %M406                 (* BLUE_TANK *)
  BLK %TM2
  LD %MW2009:X0
  AND %M406               (* BLUE_TANK *)
  IN
  OUT_BLK
  LD Q
  ST %M60
  S %M407                 (* EXTRA_TIME_BLUE_TANK *)
  END_BLK
  BLK %TM3
  LD %MW2009:X0
  AND %M407               (* EXTRA_TIME_BLUE_TANK *)
  IN
  OUT_BLK
  LD Q
  R %M406                 (* BLUE_TANK *)
  R %M407                 (* EXTRA_TIME_BLUE_TANK *)
  END_BLK
  LD %MW2009:X0
  ANDF %M19
  S %M408                 (* GREEN_TANK *)
  BLK %TM4
  LD %MW2009:X0
  AND %M408               (* GREEN_TANK *)
  IN
  OUT_BLK
  LD Q
  ST %M61
  S %M409                 (* EXTRA_TIME_GREEN_TANK *)
  END_BLK
  BLK %TM5
  LD %MW2009:X0
  AND %M409               (* EXTRA_TIME_GREEN_TANK *)
  IN
  OUT_BLK
  LD Q
  R %M408                 (* GREEN_TANK *)
  R %M409                 (* EXTRA_TIME_GREEN_TANK *)
  END_BLK
  MULTIFB
  // as ST:
  //   IF FALLING(%M18) THEN BLUE_TANK := TRUE; END_IF;
  //   %TM2(IN := BLUE_TANK);
  //   %M60 := %TM2.Q;
  //   IF %TM2.Q THEN EXTRA_TIME_BLUE_TANK := TRUE; END_IF;
  //   %TM3(IN := EXTRA_TIME_BLUE_TANK);
  //   IF %TM3.Q THEN BLUE_TANK := FALSE; END_IF;
  //   IF %TM3.Q THEN EXTRA_TIME_BLUE_TANK := FALSE; END_IF;
  //   IF FALLING(%M19) THEN GREEN_TANK := TRUE; END_IF;
  //   %TM4(IN := GREEN_TANK);
  //   %M61 := %TM4.Q;
  //   IF %TM4.Q THEN EXTRA_TIME_GREEN_TANK := TRUE; END_IF;
  //   %TM5(IN := EXTRA_TIME_GREEN_TANK);
  //   IF %TM5.Q THEN GREEN_TANK := FALSE; END_IF;
  //   IF %TM5.Q THEN EXTRA_TIME_GREEN_TANK := FALSE; END_IF;

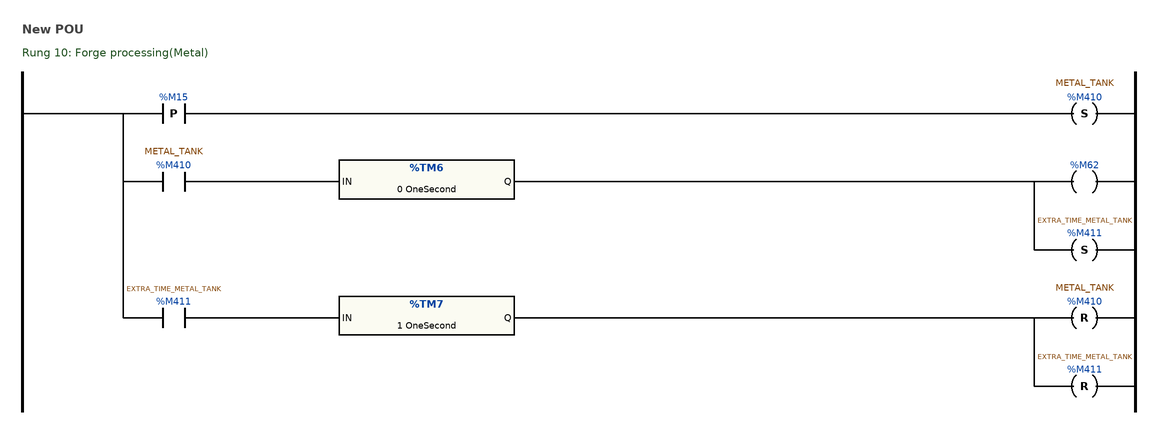

// Rung 10: Forge processing(Metal)
  LD 1
  MULTIFB
  LD 1
  ST %MW2009:X0
  LD %MW2009:X0
  ANDR %M15
  S %M410                 (* METAL_TANK *)
  BLK %TM6
  LD %MW2009:X0
  AND %M410               (* METAL_TANK *)
  IN
  OUT_BLK
  LD Q
  ST %M62
  S %M411                 (* EXTRA_TIME_METAL_TANK *)
  END_BLK
  BLK %TM7
  LD %MW2009:X0
  AND %M411               (* EXTRA_TIME_METAL_TANK *)
  IN
  OUT_BLK
  LD Q
  R %M410                 (* METAL_TANK *)
  R %M411                 (* EXTRA_TIME_METAL_TANK *)
  END_BLK
  MULTIFB
  // as ST:
  //   IF RISING(%M15) THEN METAL_TANK := TRUE; END_IF;
  //   %TM6(IN := METAL_TANK);
  //   %M62 := %TM6.Q;
  //   IF %TM6.Q THEN EXTRA_TIME_METAL_TANK := TRUE; END_IF;
  //   %TM7(IN := EXTRA_TIME_METAL_TANK);
  //   IF %TM7.Q THEN METAL_TANK := FALSE; END_IF;
  //   IF %TM7.Q THEN EXTRA_TIME_METAL_TANK := FALSE; END_IF;

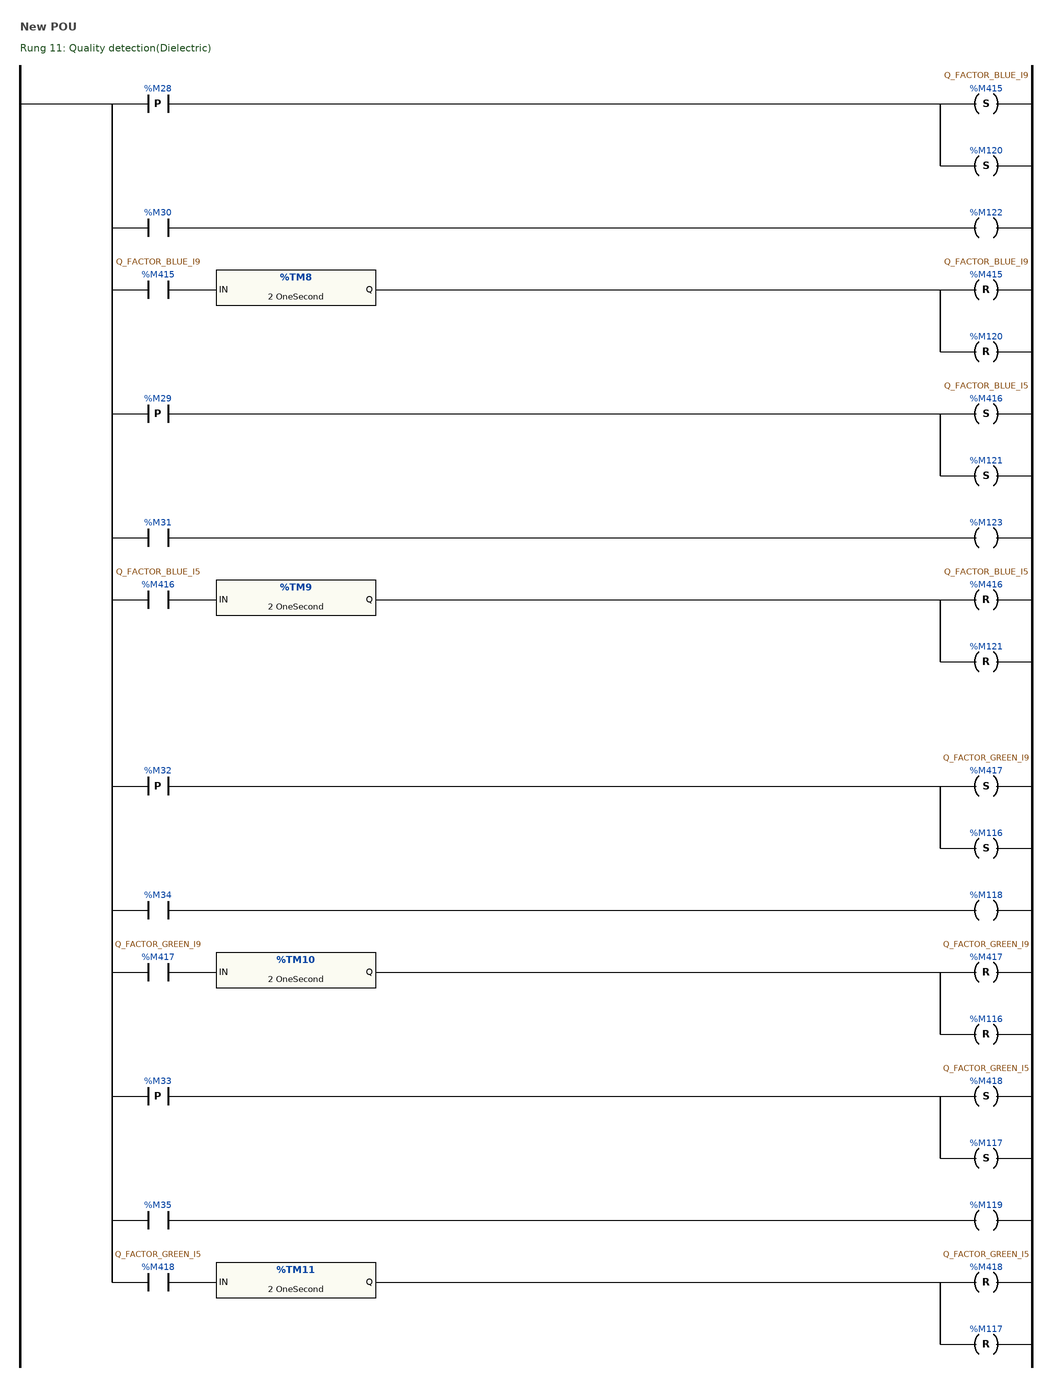

// Rung 11: Quality detection(Dielectric)
  LD 1
  MULTIFB
  LD 1
  ST %MW2009:X0
  LD %MW2009:X0
  MPS
  ANDR %M28
  S %M415                 (* Q_FACTOR_BLUE_I9 *)
  S %M120
  MPP
  AND %M30
  ST %M122
  BLK %TM8
  LD %MW2009:X0
  AND %M415               (* Q_FACTOR_BLUE_I9 *)
  IN
  OUT_BLK
  LD Q
  R %M415                 (* Q_FACTOR_BLUE_I9 *)
  R %M120
  END_BLK
  LD %MW2009:X0
  MPS
  ANDR %M29
  S %M416                 (* Q_FACTOR_BLUE_I5 *)
  S %M121
  MPP
  AND %M31
  ST %M123
  BLK %TM9
  LD %MW2009:X0
  AND %M416               (* Q_FACTOR_BLUE_I5 *)
  IN
  OUT_BLK
  LD Q
  R %M416                 (* Q_FACTOR_BLUE_I5 *)
  R %M121
  END_BLK
  LD %MW2009:X0
  MPS
  ANDR %M32
  S %M417                 (* Q_FACTOR_GREEN_I9 *)
  S %M116
  MPP
  AND %M34
  ST %M118
  BLK %TM10
  LD %MW2009:X0
  AND %M417               (* Q_FACTOR_GREEN_I9 *)
  IN
  OUT_BLK
  LD Q
  R %M417                 (* Q_FACTOR_GREEN_I9 *)
  R %M116
  END_BLK
  LD %MW2009:X0
  MPS
  ANDR %M33
  S %M418                 (* Q_FACTOR_GREEN_I5 *)
  S %M117
  MPP
  AND %M35
  ST %M119
  BLK %TM11
  LD %MW2009:X0
  AND %M418               (* Q_FACTOR_GREEN_I5 *)
  IN
  OUT_BLK
  LD Q
  R %M418                 (* Q_FACTOR_GREEN_I5 *)
  R %M117
  END_BLK
  MULTIFB
  // as ST:
  //   IF RISING(%M28) THEN Q_FACTOR_BLUE_I9 := TRUE; END_IF;
  //   IF RISING(%M28) THEN %M120 := TRUE; END_IF;
  //   %M122 := %M30;
  //   %TM8(IN := Q_FACTOR_BLUE_I9);
  //   IF %TM8.Q THEN Q_FACTOR_BLUE_I9 := FALSE; END_IF;
  //   IF %TM8.Q THEN %M120 := FALSE; END_IF;
  //   IF RISING(%M29) THEN Q_FACTOR_BLUE_I5 := TRUE; END_IF;
  //   IF RISING(%M29) THEN %M121 := TRUE; END_IF;
  //   %M123 := %M31;
  //   %TM9(IN := Q_FACTOR_BLUE_I5);
  //   IF %TM9.Q THEN Q_FACTOR_BLUE_I5 := FALSE; END_IF;
  //   IF %TM9.Q THEN %M121 := FALSE; END_IF;
  //   IF RISING(%M32) THEN Q_FACTOR_GREEN_I9 := TRUE; END_IF;
  //   IF RISING(%M32) THEN %M116 := TRUE; END_IF;
  //   %M118 := %M34;
  //   %TM10(IN := Q_FACTOR_GREEN_I9);
  //   IF %TM10.Q THEN Q_FACTOR_GREEN_I9 := FALSE; END_IF;
  //   IF %TM10.Q THEN %M116 := FALSE; END_IF;
  //   IF RISING(%M33) THEN Q_FACTOR_GREEN_I5 := TRUE; END_IF;
  //   IF RISING(%M33) THEN %M117 := TRUE; END_IF;
  //   %M119 := %M35;
  //   %TM11(IN := Q_FACTOR_GREEN_I5);
  //   IF %TM11.Q THEN Q_FACTOR_GREEN_I5 := FALSE; END_IF;
  //   IF %TM11.Q THEN %M117 := FALSE; END_IF;

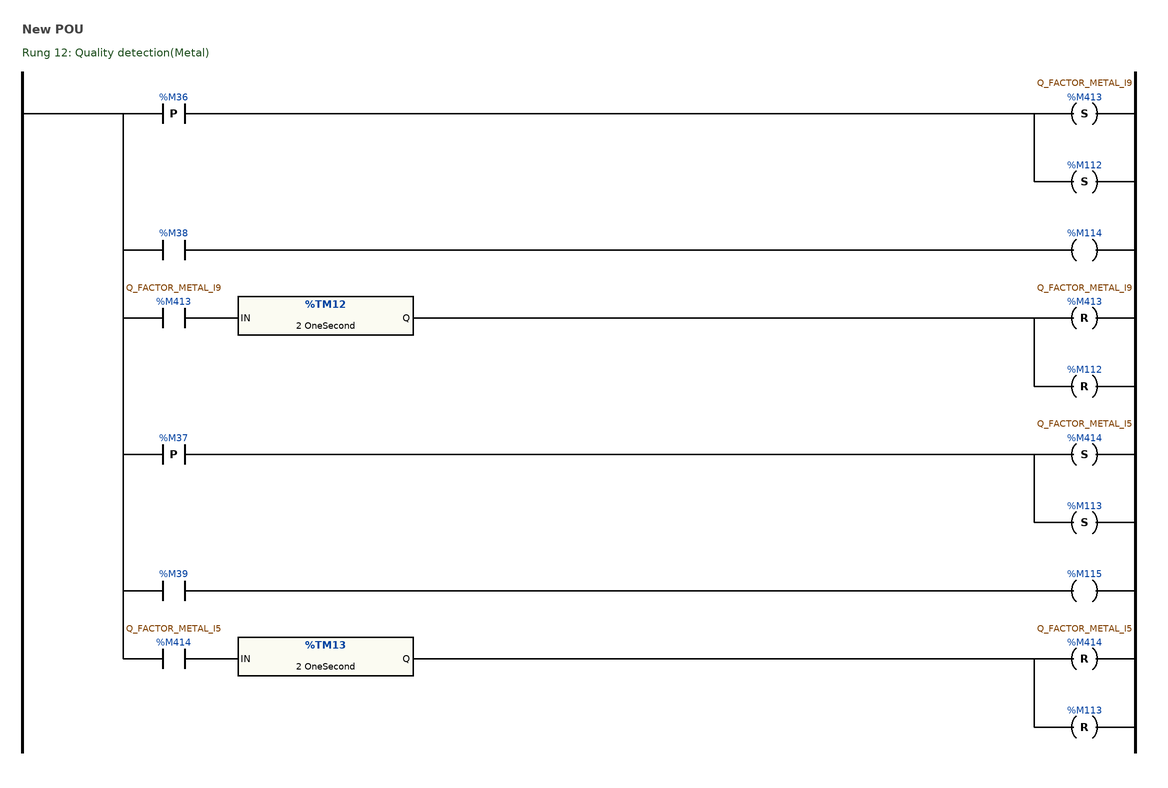

// Rung 12: Quality detection(Metal)
  LD 1
  MULTIFB
  LD 1
  ST %MW2009:X0
  LD %MW2009:X0
  MPS
  ANDR %M36
  S %M413                 (* Q_FACTOR_METAL_I9 *)
  S %M112
  MPP
  AND %M38
  ST %M114
  BLK %TM12
  LD %MW2009:X0
  AND %M413               (* Q_FACTOR_METAL_I9 *)
  IN
  OUT_BLK
  LD Q
  R %M413                 (* Q_FACTOR_METAL_I9 *)
  R %M112
  END_BLK
  LD %MW2009:X0
  MPS
  ANDR %M37
  S %M414                 (* Q_FACTOR_METAL_I5 *)
  S %M113
  MPP
  AND %M39
  ST %M115
  BLK %TM13
  LD %MW2009:X0
  AND %M414               (* Q_FACTOR_METAL_I5 *)
  IN
  OUT_BLK
  LD Q
  R %M414                 (* Q_FACTOR_METAL_I5 *)
  R %M113
  END_BLK
  MULTIFB
  // as ST:
  //   IF RISING(%M36) THEN Q_FACTOR_METAL_I9 := TRUE; END_IF;
  //   IF RISING(%M36) THEN %M112 := TRUE; END_IF;
  //   %M114 := %M38;
  //   %TM12(IN := Q_FACTOR_METAL_I9);
  //   IF %TM12.Q THEN Q_FACTOR_METAL_I9 := FALSE; END_IF;
  //   IF %TM12.Q THEN %M112 := FALSE; END_IF;
  //   IF RISING(%M37) THEN Q_FACTOR_METAL_I5 := TRUE; END_IF;
  //   IF RISING(%M37) THEN %M113 := TRUE; END_IF;
  //   %M115 := %M39;
  //   %TM13(IN := Q_FACTOR_METAL_I5);
  //   IF %TM13.Q THEN Q_FACTOR_METAL_I5 := FALSE; END_IF;
  //   IF %TM13.Q THEN %M113 := FALSE; END_IF;

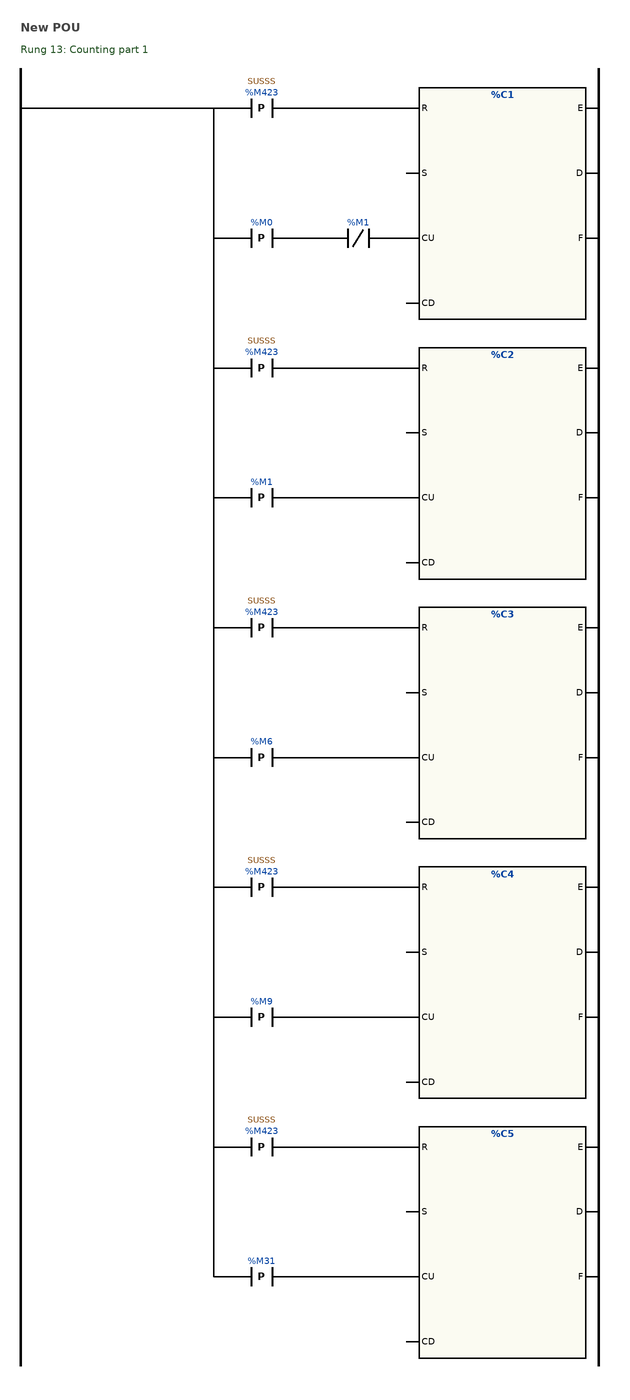

// Rung 13: Counting part 1
  LD 1
  MULTIFB
  LD 1
  ST %MW2009:X0
  BLK %C1
  LD %MW2009:X0
  MPS
  ANDR %M423              (* SUSSS *)
  R
  MPP
  ANDR %M0
  ANDN %M1
  CU
  END_BLK
  BLK %C2
  LD %MW2009:X0
  MPS
  ANDR %M423              (* SUSSS *)
  R
  MPP
  ANDR %M1
  CU
  END_BLK
  BLK %C3
  LD %MW2009:X0
  MPS
  ANDR %M423              (* SUSSS *)
  R
  MPP
  ANDR %M6
  CU
  END_BLK
  BLK %C4
  LD %MW2009:X0
  MPS
  ANDR %M423              (* SUSSS *)
  R
  MPP
  ANDR %M9
  CU
  END_BLK
  BLK %C5
  LD %MW2009:X0
  MPS
  ANDR %M423              (* SUSSS *)
  R
  MPP
  ANDR %M31
  CU
  END_BLK
  MULTIFB
  // as ST:
  //   %C1(R := RISING(SUSSS), CU := RISING(%M0) AND NOT %M1);
  //   %C2(R := RISING(SUSSS), CU := RISING(%M1));
  //   %C3(R := RISING(SUSSS), CU := RISING(%M6));
  //   %C4(R := RISING(SUSSS), CU := RISING(%M9));
  //   %C5(R := RISING(SUSSS), CU := RISING(%M31));

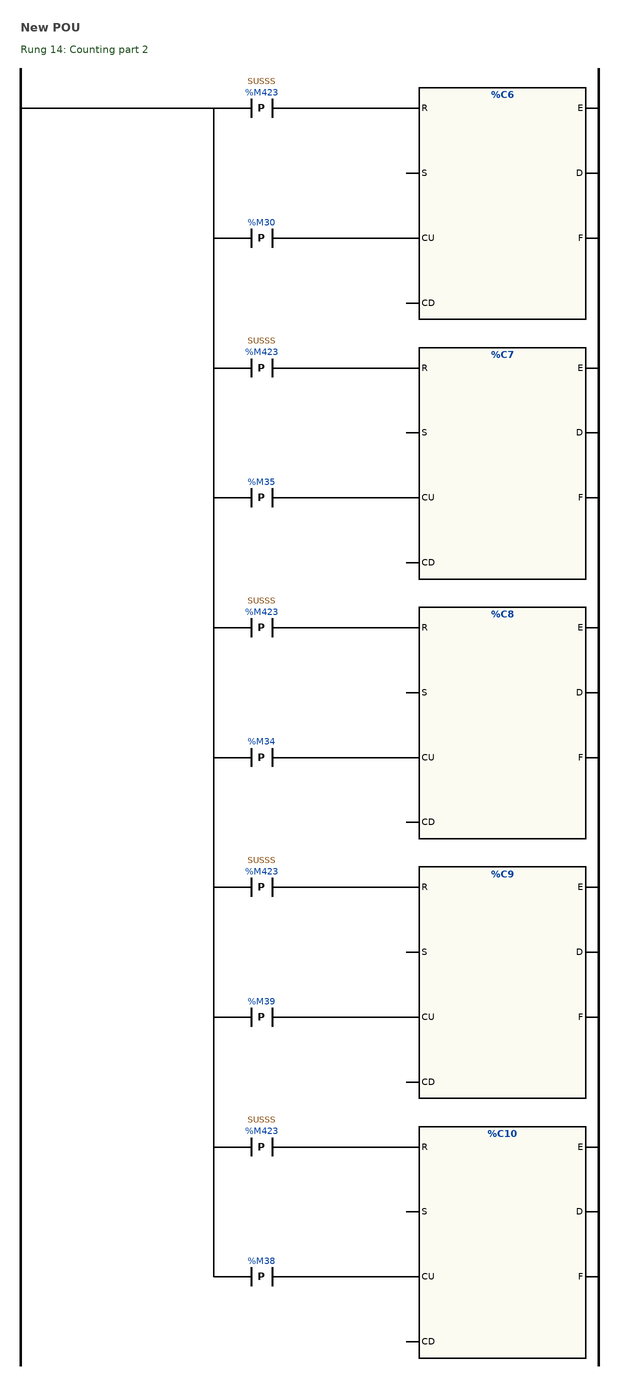

// Rung 14: Counting part 2
  LD 1
  MULTIFB
  LD 1
  ST %MW2009:X0
  BLK %C6
  LD %MW2009:X0
  MPS
  ANDR %M423              (* SUSSS *)
  R
  MPP
  ANDR %M30
  CU
  END_BLK
  BLK %C7
  LD %MW2009:X0
  MPS
  ANDR %M423              (* SUSSS *)
  R
  MPP
  ANDR %M35
  CU
  END_BLK
  BLK %C8
  LD %MW2009:X0
  MPS
  ANDR %M423              (* SUSSS *)
  R
  MPP
  ANDR %M34
  CU
  END_BLK
  BLK %C9
  LD %MW2009:X0
  MPS
  ANDR %M423              (* SUSSS *)
  R
  MPP
  ANDR %M39
  CU
  END_BLK
  BLK %C10
  LD %MW2009:X0
  MPS
  ANDR %M423              (* SUSSS *)
  R
  MPP
  ANDR %M38
  CU
  END_BLK
  MULTIFB
  // as ST:
  //   %C6(R := RISING(SUSSS), CU := RISING(%M30));
  //   %C7(R := RISING(SUSSS), CU := RISING(%M35));
  //   %C8(R := RISING(SUSSS), CU := RISING(%M34));
  //   %C9(R := RISING(SUSSS), CU := RISING(%M39));
  //   %C10(R := RISING(SUSSS), CU := RISING(%M38));

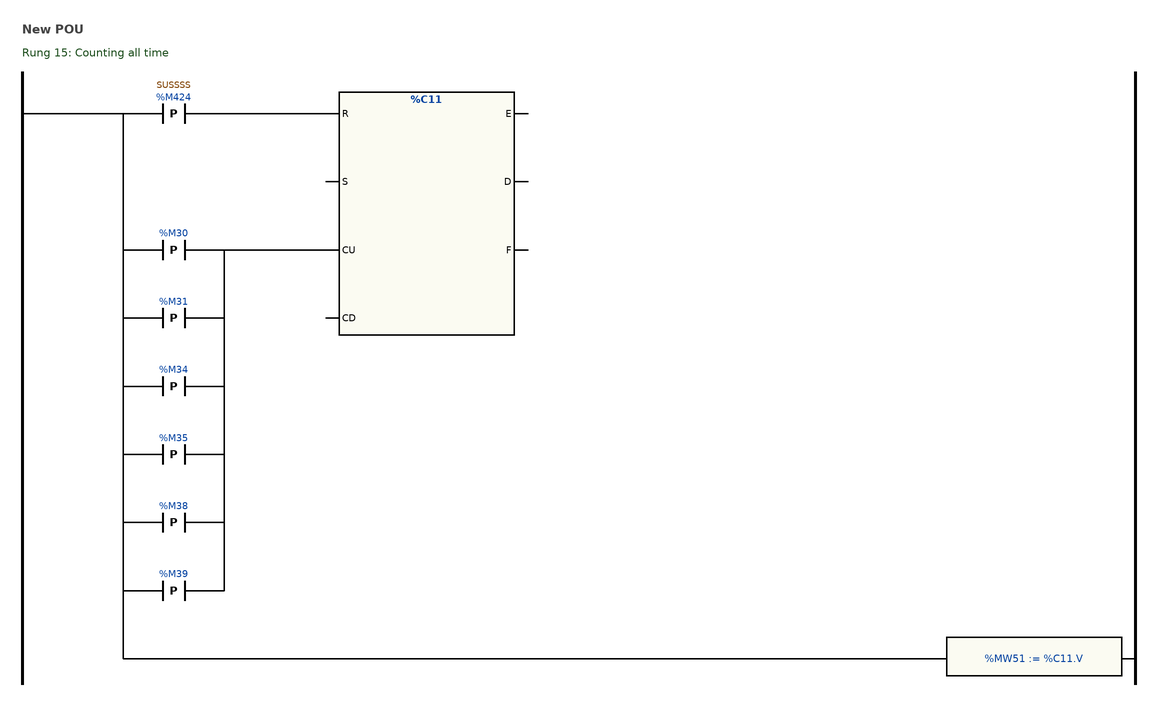

// Rung 15: Counting all time
  LD 1
  MULTIFB
  LD 1
  ST %MW2009:X0
  BLK %C11
  LD %MW2009:X0
  MPS
  ANDR %M424              (* SUSSSS *)
  R
  MPP
  AND(R %M30
  ORR %M31
  ORR %M34
  ORR %M35
  ORR %M38
  ORR %M39
  )
  CU
  END_BLK
  LD %MW2009:X0
  [ %MW51 := %C11.V ]
  MULTIFB
  // as ST:
  //   %C11(R := RISING(SUSSSS), CU := RISING(%M30) OR RISING(%M31) OR RISING(%M34) OR RISING(%M35) OR RISING(%M38) OR RISING(%M39));
  //   %MW51 := %C11.V;

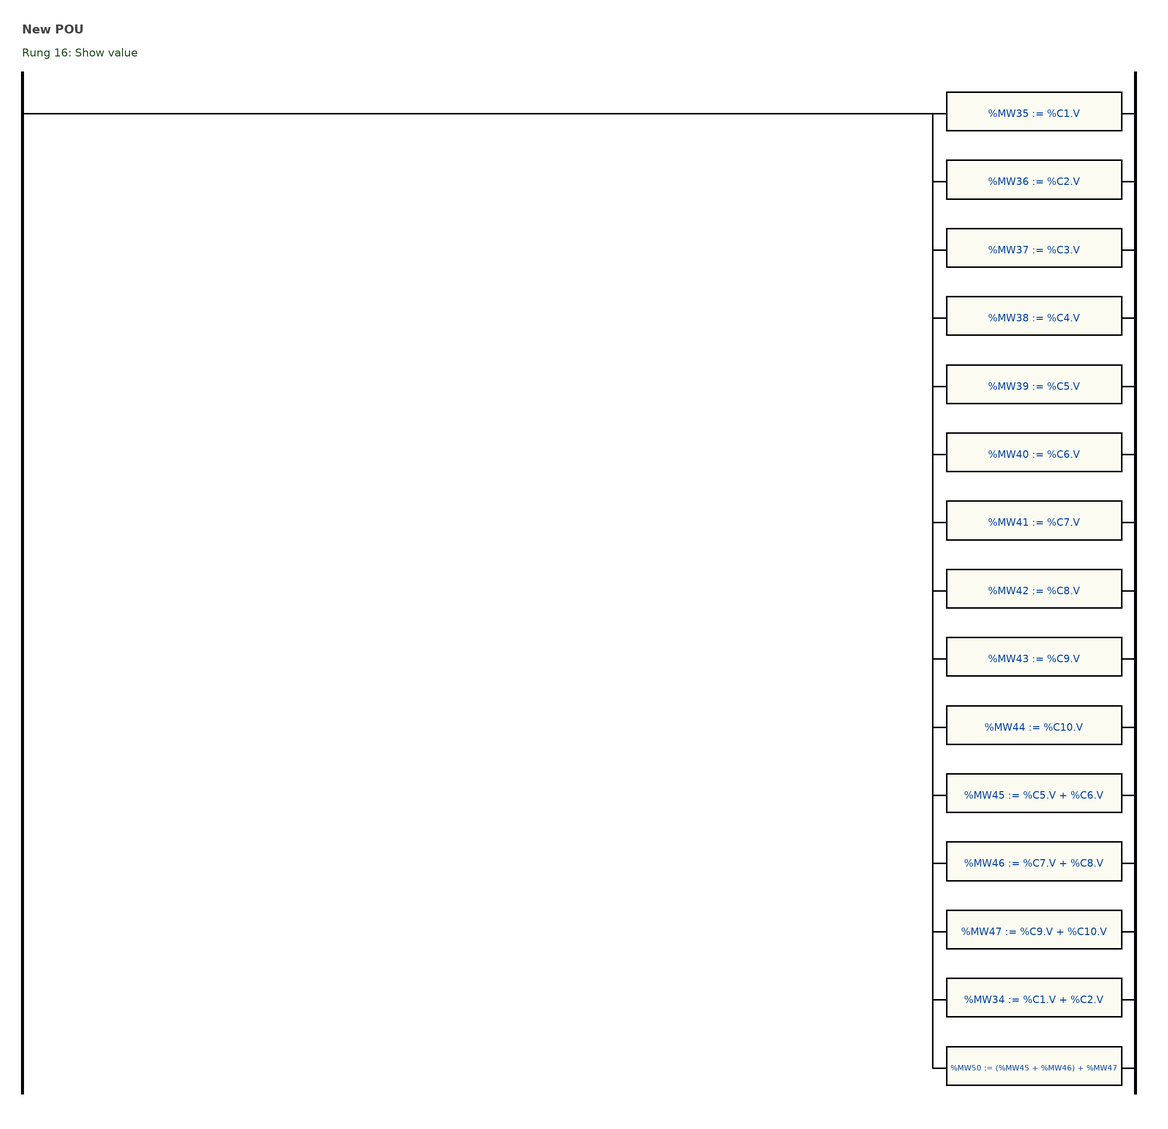

// Rung 16: Show value
  LD 1
  [ %MW35 := %C1.V ]
  [ %MW36 := %C2.V ]
  [ %MW37 := %C3.V ]
  [ %MW38 := %C4.V ]
  [ %MW39 := %C5.V ]
  [ %MW40 := %C6.V ]
  [ %MW41 := %C7.V ]
  [ %MW42 := %C8.V ]
  [ %MW43 := %C9.V ]
  [ %MW44 := %C10.V ]
  [ %MW45 := %C5.V + %C6.V ]
  [ %MW46 := %C7.V + %C8.V ]
  [ %MW47 := %C9.V + %C10.V ]
  [ %MW34 := %C1.V + %C2.V ]
  [ %MW50 := ( %MW45 + %MW46 ) + %MW47 ]
  // as ST:
  //   %MW35 := %C1.V;
  //   %MW36 := %C2.V;
  //   %MW37 := %C3.V;
  //   %MW38 := %C4.V;
  //   %MW39 := %C5.V;
  //   %MW40 := %C6.V;
  //   %MW41 := %C7.V;
  //   %MW42 := %C8.V;
  //   %MW43 := %C9.V;
  //   %MW44 := %C10.V;
  //   %MW45 := %C5.V + %C6.V;
  //   %MW46 := %C7.V + %C8.V;
  //   %MW47 := %C9.V + %C10.V;
  //   %MW34 := %C1.V + %C2.V;
  //   %MW50 := ( %MW45 + %MW46 ) + %MW47;

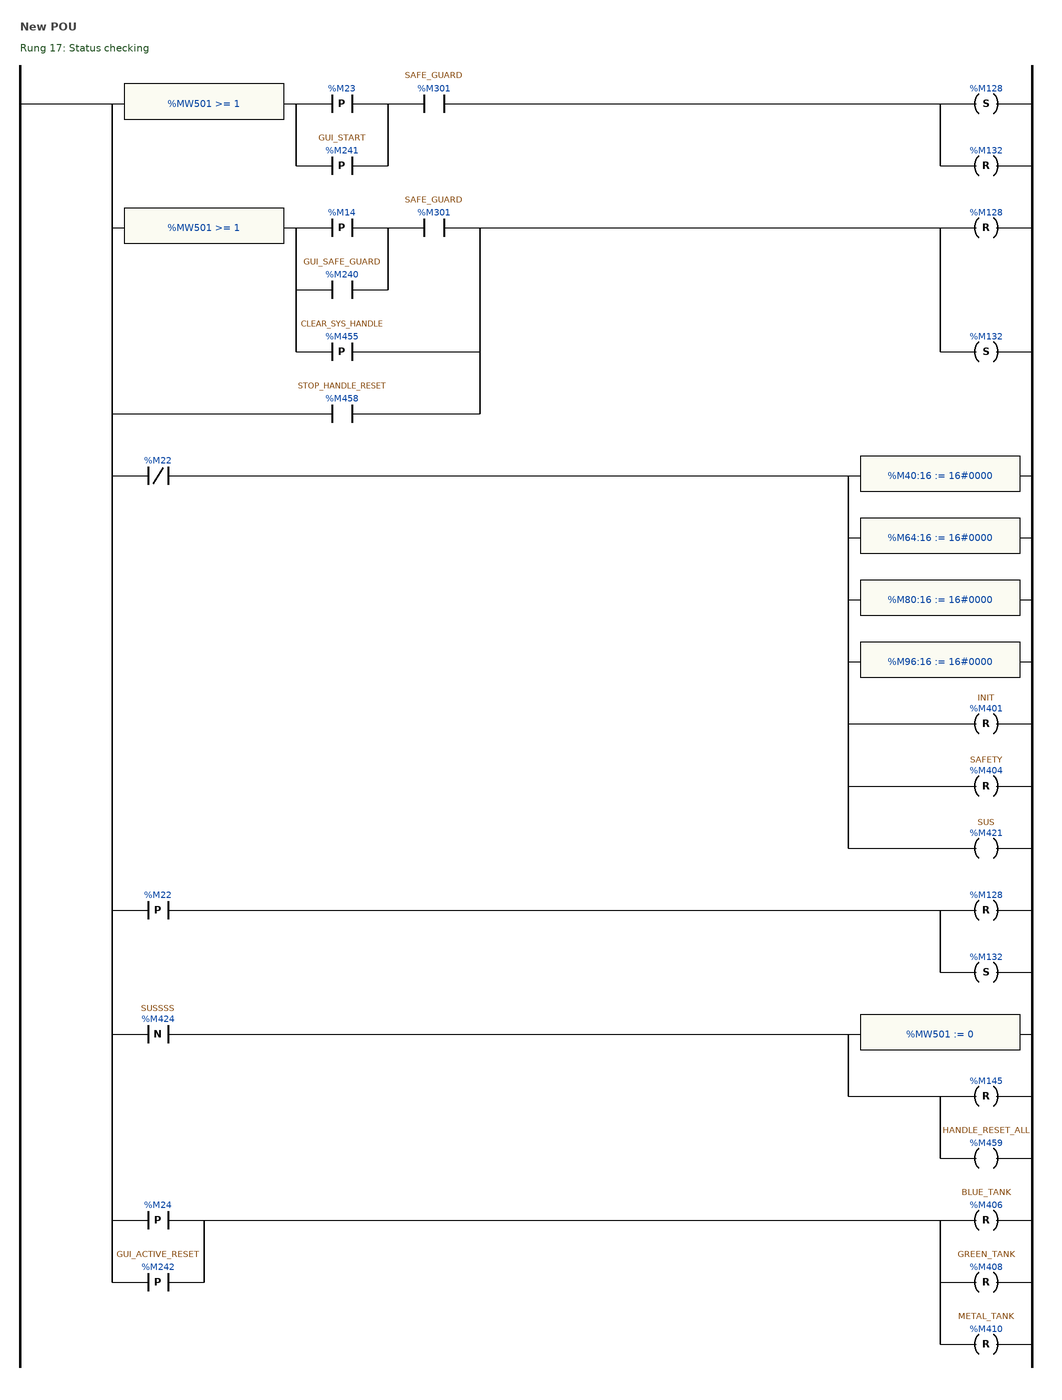

// Rung 17: Status checking
  LD 1
  MPS
  AND [ %MW501 >= 1 ]
  AND(R %M23
  ORR %M241               (* GUI_START *)
  )
  AND %M301               (* SAFE_GUARD *)
  S %M128
  R %M132
  MRD
  AND( [ %MW501 >= 1 ]
  AND(R %M14
  OR %M240                (* GUI_SAFE_GUARD *)
  AND %M301               (* SAFE_GUARD *)
  ORR %M455               (* CLEAR_SYS_HANDLE *)
  )
  OR %M458                (* STOP_HANDLE_RESET *)
  )
  R %M128
  S %M132
  MRD
  ANDN %M22
  [ %M40:16 := 16#0000 ]
  [ %M64:16 := 16#0000 ]
  [ %M80:16 := 16#0000 ]
  [ %M96:16 := 16#0000 ]
  R %M401                 (* INIT *)
  R %M404                 (* SAFETY *)
  ST %M421                (* SUS *)
  MRD
  ANDR %M22
  R %M128
  S %M132
  MRD
  ANDF %M424              (* SUSSSS *)
  [ %MW501 := 0 ]
  R %M145
  ST %M459                (* HANDLE_RESET_ALL *)
  MPP
  AND(R %M24
  ORR %M242               (* GUI_ACTIVE_RESET *)
  )
  R %M406                 (* BLUE_TANK *)
  R %M408                 (* GREEN_TANK *)
  R %M410                 (* METAL_TANK *)
  // as ST:
  //   IF %MW501 >= 1 AND (RISING(%M23) OR RISING(GUI_START)) AND SAFE_GUARD THEN %M128 := TRUE; END_IF;
  //   IF %MW501 >= 1 AND (RISING(%M23) OR RISING(GUI_START)) AND SAFE_GUARD THEN %M132 := FALSE; END_IF;
  //   IF %MW501 >= 1 AND ((RISING(%M14) OR GUI_SAFE_GUARD) AND SAFE_GUARD OR RISING(CLEAR_SYS_HANDLE)) OR STOP_HANDLE_RESET THEN %M128 := FALSE; END_IF;
  //   IF %MW501 >= 1 AND ((RISING(%M14) OR GUI_SAFE_GUARD) AND SAFE_GUARD OR RISING(CLEAR_SYS_HANDLE)) OR STOP_HANDLE_RESET THEN %M132 := TRUE; END_IF;
  //   IF NOT %M22 THEN %M40:16 := 16#0000; END_IF;
  //   IF NOT %M22 THEN %M64:16 := 16#0000; END_IF;
  //   IF NOT %M22 THEN %M80:16 := 16#0000; END_IF;
  //   IF NOT %M22 THEN %M96:16 := 16#0000; END_IF;
  //   IF NOT %M22 THEN INIT := FALSE; END_IF;
  //   IF NOT %M22 THEN SAFETY := FALSE; END_IF;
  //   SUS := NOT %M22;
  //   IF RISING(%M22) THEN %M128 := FALSE; END_IF;
  //   IF RISING(%M22) THEN %M132 := TRUE; END_IF;
  //   IF FALLING(SUSSSS) THEN %MW501 := 0; END_IF;
  //   IF FALLING(SUSSSS) THEN %M145 := FALSE; END_IF;
  //   HANDLE_RESET_ALL := FALLING(SUSSSS);
  //   IF RISING(%M24) OR RISING(GUI_ACTIVE_RESET) THEN BLUE_TANK := FALSE; END_IF;
  //   IF RISING(%M24) OR RISING(GUI_ACTIVE_RESET) THEN GREEN_TANK := FALSE; END_IF;
  //   IF RISING(%M24) OR RISING(GUI_ACTIVE_RESET) THEN METAL_TANK := FALSE; END_IF;

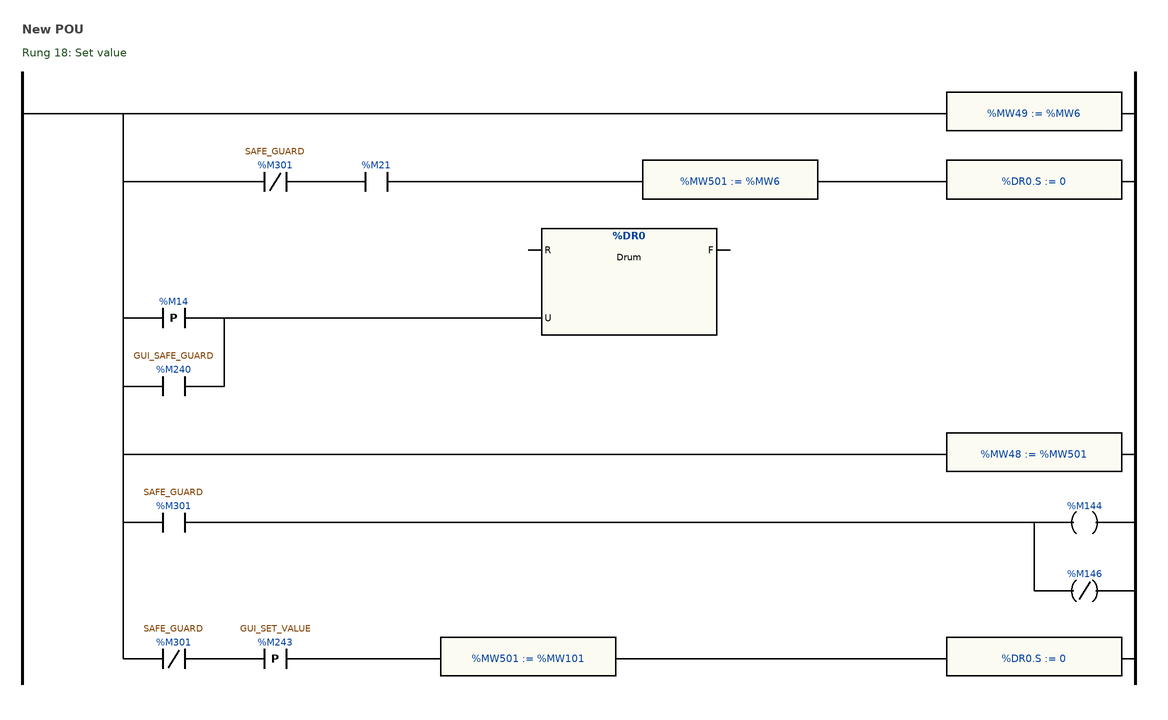

// Rung 18: Set value
  LD 1
  MULTIFB
  LD 1
  ST %MW2009:X0
  LD %MW2009:X0
  MPS
  [ %MW49 := %MW6 ]
  MPP
  ANDN %M301              (* SAFE_GUARD *)
  AND %M21
  OPER [ %MW501 := %MW6 ]
  [ %DR0.S := 0 ]
  BLK %DR0
  LD %MW2009:X0
  AND(R %M14
  OR %M240                (* GUI_SAFE_GUARD *)
  )
  U
  END_BLK
  LD %MW2009:X0
  MPS
  [ %MW48 := %MW501 ]
  MRD
  AND %M301               (* SAFE_GUARD *)
  ST %M144
  STN %M146
  MPP
  ANDN %M301              (* SAFE_GUARD *)
  ANDR %M243              (* GUI_SET_VALUE *)
  OPER [ %MW501 := %MW101 ]
  [ %DR0.S := 0 ]
  MULTIFB
  // as ST:
  //   %MW49 := %MW6;
  //   IF NOT SAFE_GUARD AND %M21 THEN %MW501 := %MW6; END_IF;
  //   IF NOT SAFE_GUARD AND %M21 THEN %DR0.S := 0; END_IF;
  //   %DR0(U := RISING(%M14) OR GUI_SAFE_GUARD);
  //   %MW48 := %MW501;
  //   %M144 := SAFE_GUARD;
  //   %M146 := NOT SAFE_GUARD;
  //   IF NOT SAFE_GUARD AND RISING(GUI_SET_VALUE) THEN %MW501 := %MW101; END_IF;
  //   IF NOT SAFE_GUARD AND RISING(GUI_SET_VALUE) THEN %DR0.S := 0; END_IF;

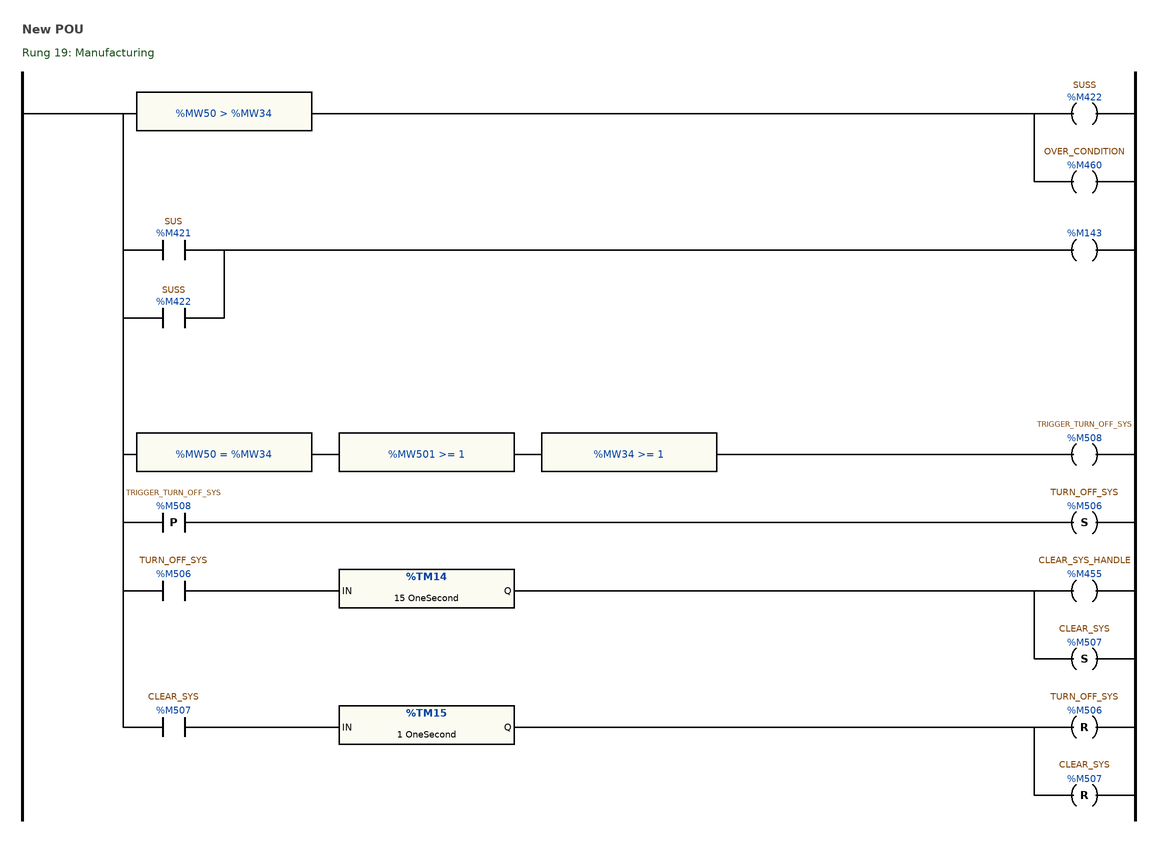

// Rung 19: Manufacturing
  LD 1
  MULTIFB
  LD 1
  ST %MW2009:X0
  LD %MW2009:X0
  MPS
  AND [ %MW50 > %MW34 ]
  ST %M422                (* SUSS *)
  ST %M460                (* OVER_CONDITION *)
  MRD
  AND( %M421              (* SUS *)
  OR %M422                (* SUSS *)
  )
  ST %M143
  MRD
  AND [ %MW50 = %MW34 ]
  AND [ %MW501 >= 1 ]
  AND [ %MW34 >= 1 ]
  ST %M508                (* TRIGGER_TURN_OFF_SYS *)
  MPP
  ANDR %M508              (* TRIGGER_TURN_OFF_SYS *)
  S %M506                 (* TURN_OFF_SYS *)
  BLK %TM14
  LD %MW2009:X0
  AND %M506               (* TURN_OFF_SYS *)
  IN
  OUT_BLK
  LD Q
  ST %M455                (* CLEAR_SYS_HANDLE *)
  S %M507                 (* CLEAR_SYS *)
  END_BLK
  BLK %TM15
  LD %MW2009:X0
  AND %M507               (* CLEAR_SYS *)
  IN
  OUT_BLK
  LD Q
  R %M506                 (* TURN_OFF_SYS *)
  R %M507                 (* CLEAR_SYS *)
  END_BLK
  MULTIFB
  // as ST:
  //   SUSS := %MW50 > %MW34;
  //   OVER_CONDITION := %MW50 > %MW34;
  //   %M143 := SUS OR SUSS;
  //   TRIGGER_TURN_OFF_SYS := %MW50 = %MW34 AND %MW501 >= 1 AND %MW34 >= 1;
  //   IF RISING(TRIGGER_TURN_OFF_SYS) THEN TURN_OFF_SYS := TRUE; END_IF;
  //   %TM14(IN := TURN_OFF_SYS);
  //   CLEAR_SYS_HANDLE := %TM14.Q;
  //   IF %TM14.Q THEN CLEAR_SYS := TRUE; END_IF;
  //   %TM15(IN := CLEAR_SYS);
  //   IF %TM15.Q THEN TURN_OFF_SYS := FALSE; END_IF;
  //   IF %TM15.Q THEN CLEAR_SYS := FALSE; END_IF;

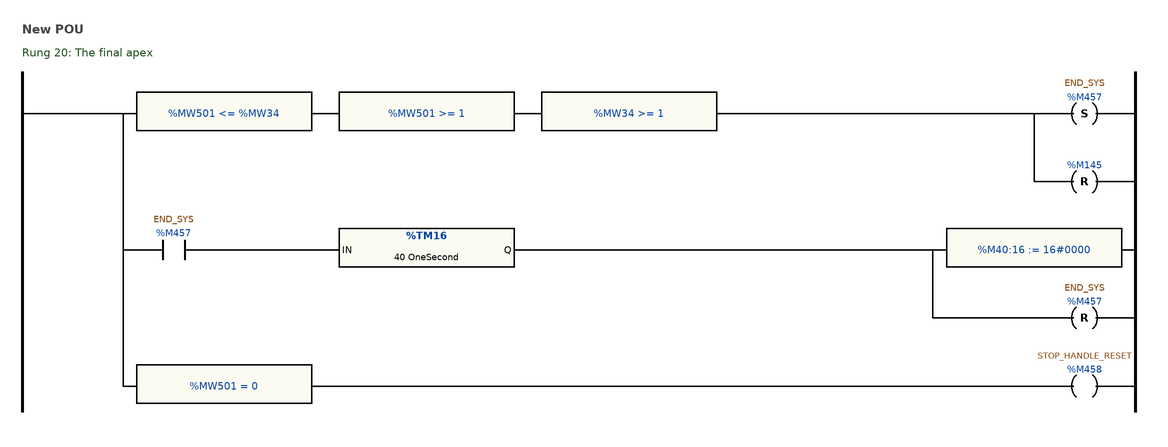

// Rung 20: The final apex
  LD 1
  MULTIFB
  LD 1
  ST %MW2009:X0
  LD %MW2009:X0
  AND [ %MW501 <= %MW34 ]
  AND [ %MW501 >= 1 ]
  AND [ %MW34 >= 1 ]
  S %M457                 (* END_SYS *)
  R %M145
  BLK %TM16
  LD %MW2009:X0
  AND %M457               (* END_SYS *)
  IN
  OUT_BLK
  LD Q
  [ %M40:16 := 16#0000 ]
  R %M457                 (* END_SYS *)
  END_BLK
  LD %MW2009:X0
  AND [ %MW501 = 0 ]
  ST %M458                (* STOP_HANDLE_RESET *)
  MULTIFB
  // as ST:
  //   IF %MW501 <= %MW34 AND %MW501 >= 1 AND %MW34 >= 1 THEN END_SYS := TRUE; END_IF;
  //   IF %MW501 <= %MW34 AND %MW501 >= 1 AND %MW34 >= 1 THEN %M145 := FALSE; END_IF;
  //   %TM16(IN := END_SYS);
  //   IF %TM16.Q THEN %M40:16 := 16#0000; END_IF;
  //   IF %TM16.Q THEN END_SYS := FALSE; END_IF;
  //   STOP_HANDLE_RESET := %MW501 = 0;
